;FOLD SLIN P513 Vel=1 m/s CPDAT513 Tool[4]:Microflown3D Base[0];%{PE}
;FOLD Parameters ;%{h}
;Params IlfProvider=kukaroboter.basistech.inlineforms.movement.spline; Kuka.IsGlobalPoint=False; Kuka.PointName=P513; Kuka.BlendingEnabled=False; Kuka.MoveDataName=CPDAT513; Kuka.VelocityPath=1.000; Kuka.VelocityFieldEnabled=True; Kuka.ColDetectFieldEnabled=True; Kuka.CurrentCDSetIndex=0; Kuka.MovementParameterFieldEnabled=True; IlfCommand=SLIN
;ENDFOLD
SLIN XP513 WITH $VEL = SVEL_CP(2.0, , LCPDAT513),$TOOL = STOOL2(FP513),$BASE = SBASE(FP513.BASE_NO),$IPO_MODE = SIPO_MODE(FP513.IPO_FRAME),$LOAD = SLOAD(FP513.TOOL_NO),$ACC = SACC_CP(LCPDAT513),$ORI_TYPE = SORI_TYP(LCPDAT513),$APO = SAPO(LCPDAT513),$JERK = SJERK(LCPDAT513),$COLLMON_TOL_PRO[1] = USE_CM_PRO_VALUES(0)
;ENDFOLD

;FOLD SLIN P514 Vel=1 m/s CPDAT514 Tool[4]:Microflown3D Base[0];%{PE}
;FOLD Parameters ;%{h}
;Params IlfProvider=kukaroboter.basistech.inlineforms.movement.spline; Kuka.IsGlobalPoint=False; Kuka.PointName=P514; Kuka.BlendingEnabled=False; Kuka.MoveDataName=CPDAT514; Kuka.VelocityPath=1.000; Kuka.VelocityFieldEnabled=True; Kuka.ColDetectFieldEnabled=True; Kuka.CurrentCDSetIndex=0; Kuka.MovementParameterFieldEnabled=True; IlfCommand=SLIN
;ENDFOLD
SLIN XP514 WITH $VEL = SVEL_CP(2.0, , LCPDAT514),$TOOL = STOOL2(FP514),$BASE = SBASE(FP514.BASE_NO),$IPO_MODE = SIPO_MODE(FP514.IPO_FRAME),$LOAD = SLOAD(FP514.TOOL_NO),$ACC = SACC_CP(LCPDAT514),$ORI_TYPE = SORI_TYP(LCPDAT514),$APO = SAPO(LCPDAT514),$JERK = SJERK(LCPDAT514),$COLLMON_TOL_PRO[1] = USE_CM_PRO_VALUES(0)
;ENDFOLD

;FOLD SLIN P515 Vel=1 m/s CPDAT515 Tool[4]:Microflown3D Base[0];%{PE}
;FOLD Parameters ;%{h}
;Params IlfProvider=kukaroboter.basistech.inlineforms.movement.spline; Kuka.IsGlobalPoint=False; Kuka.PointName=P515; Kuka.BlendingEnabled=False; Kuka.MoveDataName=CPDAT515; Kuka.VelocityPath=1.000; Kuka.VelocityFieldEnabled=True; Kuka.ColDetectFieldEnabled=True; Kuka.CurrentCDSetIndex=0; Kuka.MovementParameterFieldEnabled=True; IlfCommand=SLIN
;ENDFOLD
SLIN XP515 WITH $VEL = SVEL_CP(2.0, , LCPDAT515),$TOOL = STOOL2(FP515),$BASE = SBASE(FP515.BASE_NO),$IPO_MODE = SIPO_MODE(FP515.IPO_FRAME),$LOAD = SLOAD(FP515.TOOL_NO),$ACC = SACC_CP(LCPDAT515),$ORI_TYPE = SORI_TYP(LCPDAT515),$APO = SAPO(LCPDAT515),$JERK = SJERK(LCPDAT515),$COLLMON_TOL_PRO[1] = USE_CM_PRO_VALUES(0)
;ENDFOLD

;FOLD SLIN P516 Vel=1 m/s CPDAT516 Tool[4]:Microflown3D Base[0];%{PE}
;FOLD Parameters ;%{h}
;Params IlfProvider=kukaroboter.basistech.inlineforms.movement.spline; Kuka.IsGlobalPoint=False; Kuka.PointName=P516; Kuka.BlendingEnabled=False; Kuka.MoveDataName=CPDAT516; Kuka.VelocityPath=1.000; Kuka.VelocityFieldEnabled=True; Kuka.ColDetectFieldEnabled=True; Kuka.CurrentCDSetIndex=0; Kuka.MovementParameterFieldEnabled=True; IlfCommand=SLIN
;ENDFOLD
SLIN XP516 WITH $VEL = SVEL_CP(2.0, , LCPDAT516),$TOOL = STOOL2(FP516),$BASE = SBASE(FP516.BASE_NO),$IPO_MODE = SIPO_MODE(FP516.IPO_FRAME),$LOAD = SLOAD(FP516.TOOL_NO),$ACC = SACC_CP(LCPDAT516),$ORI_TYPE = SORI_TYP(LCPDAT516),$APO = SAPO(LCPDAT516),$JERK = SJERK(LCPDAT516),$COLLMON_TOL_PRO[1] = USE_CM_PRO_VALUES(0)
;ENDFOLD

;FOLD SLIN P517 Vel=1 m/s CPDAT517 Tool[4]:Microflown3D Base[0];%{PE}
;FOLD Parameters ;%{h}
;Params IlfProvider=kukaroboter.basistech.inlineforms.movement.spline; Kuka.IsGlobalPoint=False; Kuka.PointName=P517; Kuka.BlendingEnabled=False; Kuka.MoveDataName=CPDAT517; Kuka.VelocityPath=1.000; Kuka.VelocityFieldEnabled=True; Kuka.ColDetectFieldEnabled=True; Kuka.CurrentCDSetIndex=0; Kuka.MovementParameterFieldEnabled=True; IlfCommand=SLIN
;ENDFOLD
SLIN XP517 WITH $VEL = SVEL_CP(2.0, , LCPDAT517),$TOOL = STOOL2(FP517),$BASE = SBASE(FP517.BASE_NO),$IPO_MODE = SIPO_MODE(FP517.IPO_FRAME),$LOAD = SLOAD(FP517.TOOL_NO),$ACC = SACC_CP(LCPDAT517),$ORI_TYPE = SORI_TYP(LCPDAT517),$APO = SAPO(LCPDAT517),$JERK = SJERK(LCPDAT517),$COLLMON_TOL_PRO[1] = USE_CM_PRO_VALUES(0)
;ENDFOLD

;FOLD SLIN P518 Vel=1 m/s CPDAT518 Tool[4]:Microflown3D Base[0];%{PE}
;FOLD Parameters ;%{h}
;Params IlfProvider=kukaroboter.basistech.inlineforms.movement.spline; Kuka.IsGlobalPoint=False; Kuka.PointName=P518; Kuka.BlendingEnabled=False; Kuka.MoveDataName=CPDAT518; Kuka.VelocityPath=1.000; Kuka.VelocityFieldEnabled=True; Kuka.ColDetectFieldEnabled=True; Kuka.CurrentCDSetIndex=0; Kuka.MovementParameterFieldEnabled=True; IlfCommand=SLIN
;ENDFOLD
SLIN XP518 WITH $VEL = SVEL_CP(2.0, , LCPDAT518),$TOOL = STOOL2(FP518),$BASE = SBASE(FP518.BASE_NO),$IPO_MODE = SIPO_MODE(FP518.IPO_FRAME),$LOAD = SLOAD(FP518.TOOL_NO),$ACC = SACC_CP(LCPDAT518),$ORI_TYPE = SORI_TYP(LCPDAT518),$APO = SAPO(LCPDAT518),$JERK = SJERK(LCPDAT518),$COLLMON_TOL_PRO[1] = USE_CM_PRO_VALUES(0)
;ENDFOLD

;FOLD SLIN P519 Vel=1 m/s CPDAT519 Tool[4]:Microflown3D Base[0];%{PE}
;FOLD Parameters ;%{h}
;Params IlfProvider=kukaroboter.basistech.inlineforms.movement.spline; Kuka.IsGlobalPoint=False; Kuka.PointName=P519; Kuka.BlendingEnabled=False; Kuka.MoveDataName=CPDAT519; Kuka.VelocityPath=1.000; Kuka.VelocityFieldEnabled=True; Kuka.ColDetectFieldEnabled=True; Kuka.CurrentCDSetIndex=0; Kuka.MovementParameterFieldEnabled=True; IlfCommand=SLIN
;ENDFOLD
SLIN XP519 WITH $VEL = SVEL_CP(2.0, , LCPDAT519),$TOOL = STOOL2(FP519),$BASE = SBASE(FP519.BASE_NO),$IPO_MODE = SIPO_MODE(FP519.IPO_FRAME),$LOAD = SLOAD(FP519.TOOL_NO),$ACC = SACC_CP(LCPDAT519),$ORI_TYPE = SORI_TYP(LCPDAT519),$APO = SAPO(LCPDAT519),$JERK = SJERK(LCPDAT519),$COLLMON_TOL_PRO[1] = USE_CM_PRO_VALUES(0)
;ENDFOLD

;FOLD SLIN P520 Vel=1 m/s CPDAT520 Tool[4]:Microflown3D Base[0];%{PE}
;FOLD Parameters ;%{h}
;Params IlfProvider=kukaroboter.basistech.inlineforms.movement.spline; Kuka.IsGlobalPoint=False; Kuka.PointName=P520; Kuka.BlendingEnabled=False; Kuka.MoveDataName=CPDAT520; Kuka.VelocityPath=1.000; Kuka.VelocityFieldEnabled=True; Kuka.ColDetectFieldEnabled=True; Kuka.CurrentCDSetIndex=0; Kuka.MovementParameterFieldEnabled=True; IlfCommand=SLIN
;ENDFOLD
SLIN XP520 WITH $VEL = SVEL_CP(2.0, , LCPDAT520),$TOOL = STOOL2(FP520),$BASE = SBASE(FP520.BASE_NO),$IPO_MODE = SIPO_MODE(FP520.IPO_FRAME),$LOAD = SLOAD(FP520.TOOL_NO),$ACC = SACC_CP(LCPDAT520),$ORI_TYPE = SORI_TYP(LCPDAT520),$APO = SAPO(LCPDAT520),$JERK = SJERK(LCPDAT520),$COLLMON_TOL_PRO[1] = USE_CM_PRO_VALUES(0)
;ENDFOLD

;FOLD SLIN P521 Vel=1 m/s CPDAT521 Tool[4]:Microflown3D Base[0];%{PE}
;FOLD Parameters ;%{h}
;Params IlfProvider=kukaroboter.basistech.inlineforms.movement.spline; Kuka.IsGlobalPoint=False; Kuka.PointName=P521; Kuka.BlendingEnabled=False; Kuka.MoveDataName=CPDAT521; Kuka.VelocityPath=1.000; Kuka.VelocityFieldEnabled=True; Kuka.ColDetectFieldEnabled=True; Kuka.CurrentCDSetIndex=0; Kuka.MovementParameterFieldEnabled=True; IlfCommand=SLIN
;ENDFOLD
SLIN XP521 WITH $VEL = SVEL_CP(2.0, , LCPDAT521),$TOOL = STOOL2(FP521),$BASE = SBASE(FP521.BASE_NO),$IPO_MODE = SIPO_MODE(FP521.IPO_FRAME),$LOAD = SLOAD(FP521.TOOL_NO),$ACC = SACC_CP(LCPDAT521),$ORI_TYPE = SORI_TYP(LCPDAT521),$APO = SAPO(LCPDAT521),$JERK = SJERK(LCPDAT521),$COLLMON_TOL_PRO[1] = USE_CM_PRO_VALUES(0)
;ENDFOLD

;FOLD SLIN P522 Vel=1 m/s CPDAT522 Tool[4]:Microflown3D Base[0];%{PE}
;FOLD Parameters ;%{h}
;Params IlfProvider=kukaroboter.basistech.inlineforms.movement.spline; Kuka.IsGlobalPoint=False; Kuka.PointName=P522; Kuka.BlendingEnabled=False; Kuka.MoveDataName=CPDAT522; Kuka.VelocityPath=1.000; Kuka.VelocityFieldEnabled=True; Kuka.ColDetectFieldEnabled=True; Kuka.CurrentCDSetIndex=0; Kuka.MovementParameterFieldEnabled=True; IlfCommand=SLIN
;ENDFOLD
SLIN XP522 WITH $VEL = SVEL_CP(2.0, , LCPDAT522),$TOOL = STOOL2(FP522),$BASE = SBASE(FP522.BASE_NO),$IPO_MODE = SIPO_MODE(FP522.IPO_FRAME),$LOAD = SLOAD(FP522.TOOL_NO),$ACC = SACC_CP(LCPDAT522),$ORI_TYPE = SORI_TYP(LCPDAT522),$APO = SAPO(LCPDAT522),$JERK = SJERK(LCPDAT522),$COLLMON_TOL_PRO[1] = USE_CM_PRO_VALUES(0)
;ENDFOLD

;FOLD SLIN P523 Vel=1 m/s CPDAT523 Tool[4]:Microflown3D Base[0];%{PE}
;FOLD Parameters ;%{h}
;Params IlfProvider=kukaroboter.basistech.inlineforms.movement.spline; Kuka.IsGlobalPoint=False; Kuka.PointName=P523; Kuka.BlendingEnabled=False; Kuka.MoveDataName=CPDAT523; Kuka.VelocityPath=1.000; Kuka.VelocityFieldEnabled=True; Kuka.ColDetectFieldEnabled=True; Kuka.CurrentCDSetIndex=0; Kuka.MovementParameterFieldEnabled=True; IlfCommand=SLIN
;ENDFOLD
SLIN XP523 WITH $VEL = SVEL_CP(2.0, , LCPDAT523),$TOOL = STOOL2(FP523),$BASE = SBASE(FP523.BASE_NO),$IPO_MODE = SIPO_MODE(FP523.IPO_FRAME),$LOAD = SLOAD(FP523.TOOL_NO),$ACC = SACC_CP(LCPDAT523),$ORI_TYPE = SORI_TYP(LCPDAT523),$APO = SAPO(LCPDAT523),$JERK = SJERK(LCPDAT523),$COLLMON_TOL_PRO[1] = USE_CM_PRO_VALUES(0)
;ENDFOLD

;FOLD SLIN P524 Vel=1 m/s CPDAT524 Tool[4]:Microflown3D Base[0];%{PE}
;FOLD Parameters ;%{h}
;Params IlfProvider=kukaroboter.basistech.inlineforms.movement.spline; Kuka.IsGlobalPoint=False; Kuka.PointName=P524; Kuka.BlendingEnabled=False; Kuka.MoveDataName=CPDAT524; Kuka.VelocityPath=1.000; Kuka.VelocityFieldEnabled=True; Kuka.ColDetectFieldEnabled=True; Kuka.CurrentCDSetIndex=0; Kuka.MovementParameterFieldEnabled=True; IlfCommand=SLIN
;ENDFOLD
SLIN XP524 WITH $VEL = SVEL_CP(2.0, , LCPDAT524),$TOOL = STOOL2(FP524),$BASE = SBASE(FP524.BASE_NO),$IPO_MODE = SIPO_MODE(FP524.IPO_FRAME),$LOAD = SLOAD(FP524.TOOL_NO),$ACC = SACC_CP(LCPDAT524),$ORI_TYPE = SORI_TYP(LCPDAT524),$APO = SAPO(LCPDAT524),$JERK = SJERK(LCPDAT524),$COLLMON_TOL_PRO[1] = USE_CM_PRO_VALUES(0)
;ENDFOLD

;FOLD SLIN P525 Vel=1 m/s CPDAT525 Tool[4]:Microflown3D Base[0];%{PE}
;FOLD Parameters ;%{h}
;Params IlfProvider=kukaroboter.basistech.inlineforms.movement.spline; Kuka.IsGlobalPoint=False; Kuka.PointName=P525; Kuka.BlendingEnabled=False; Kuka.MoveDataName=CPDAT525; Kuka.VelocityPath=1.000; Kuka.VelocityFieldEnabled=True; Kuka.ColDetectFieldEnabled=True; Kuka.CurrentCDSetIndex=0; Kuka.MovementParameterFieldEnabled=True; IlfCommand=SLIN
;ENDFOLD
SLIN XP525 WITH $VEL = SVEL_CP(2.0, , LCPDAT525),$TOOL = STOOL2(FP525),$BASE = SBASE(FP525.BASE_NO),$IPO_MODE = SIPO_MODE(FP525.IPO_FRAME),$LOAD = SLOAD(FP525.TOOL_NO),$ACC = SACC_CP(LCPDAT525),$ORI_TYPE = SORI_TYP(LCPDAT525),$APO = SAPO(LCPDAT525),$JERK = SJERK(LCPDAT525),$COLLMON_TOL_PRO[1] = USE_CM_PRO_VALUES(0)
;ENDFOLD

;FOLD SLIN P526 Vel=1 m/s CPDAT526 Tool[4]:Microflown3D Base[0];%{PE}
;FOLD Parameters ;%{h}
;Params IlfProvider=kukaroboter.basistech.inlineforms.movement.spline; Kuka.IsGlobalPoint=False; Kuka.PointName=P526; Kuka.BlendingEnabled=False; Kuka.MoveDataName=CPDAT526; Kuka.VelocityPath=1.000; Kuka.VelocityFieldEnabled=True; Kuka.ColDetectFieldEnabled=True; Kuka.CurrentCDSetIndex=0; Kuka.MovementParameterFieldEnabled=True; IlfCommand=SLIN
;ENDFOLD
SLIN XP526 WITH $VEL = SVEL_CP(2.0, , LCPDAT526),$TOOL = STOOL2(FP526),$BASE = SBASE(FP526.BASE_NO),$IPO_MODE = SIPO_MODE(FP526.IPO_FRAME),$LOAD = SLOAD(FP526.TOOL_NO),$ACC = SACC_CP(LCPDAT526),$ORI_TYPE = SORI_TYP(LCPDAT526),$APO = SAPO(LCPDAT526),$JERK = SJERK(LCPDAT526),$COLLMON_TOL_PRO[1] = USE_CM_PRO_VALUES(0)
;ENDFOLD

;FOLD SLIN P527 Vel=1 m/s CPDAT527 Tool[4]:Microflown3D Base[0];%{PE}
;FOLD Parameters ;%{h}
;Params IlfProvider=kukaroboter.basistech.inlineforms.movement.spline; Kuka.IsGlobalPoint=False; Kuka.PointName=P527; Kuka.BlendingEnabled=False; Kuka.MoveDataName=CPDAT527; Kuka.VelocityPath=1.000; Kuka.VelocityFieldEnabled=True; Kuka.ColDetectFieldEnabled=True; Kuka.CurrentCDSetIndex=0; Kuka.MovementParameterFieldEnabled=True; IlfCommand=SLIN
;ENDFOLD
SLIN XP527 WITH $VEL = SVEL_CP(2.0, , LCPDAT527),$TOOL = STOOL2(FP527),$BASE = SBASE(FP527.BASE_NO),$IPO_MODE = SIPO_MODE(FP527.IPO_FRAME),$LOAD = SLOAD(FP527.TOOL_NO),$ACC = SACC_CP(LCPDAT527),$ORI_TYPE = SORI_TYP(LCPDAT527),$APO = SAPO(LCPDAT527),$JERK = SJERK(LCPDAT527),$COLLMON_TOL_PRO[1] = USE_CM_PRO_VALUES(0)
;ENDFOLD

;FOLD SLIN P528 Vel=1 m/s CPDAT528 Tool[4]:Microflown3D Base[0];%{PE}
;FOLD Parameters ;%{h}
;Params IlfProvider=kukaroboter.basistech.inlineforms.movement.spline; Kuka.IsGlobalPoint=False; Kuka.PointName=P528; Kuka.BlendingEnabled=False; Kuka.MoveDataName=CPDAT528; Kuka.VelocityPath=1.000; Kuka.VelocityFieldEnabled=True; Kuka.ColDetectFieldEnabled=True; Kuka.CurrentCDSetIndex=0; Kuka.MovementParameterFieldEnabled=True; IlfCommand=SLIN
;ENDFOLD
SLIN XP528 WITH $VEL = SVEL_CP(2.0, , LCPDAT528),$TOOL = STOOL2(FP528),$BASE = SBASE(FP528.BASE_NO),$IPO_MODE = SIPO_MODE(FP528.IPO_FRAME),$LOAD = SLOAD(FP528.TOOL_NO),$ACC = SACC_CP(LCPDAT528),$ORI_TYPE = SORI_TYP(LCPDAT528),$APO = SAPO(LCPDAT528),$JERK = SJERK(LCPDAT528),$COLLMON_TOL_PRO[1] = USE_CM_PRO_VALUES(0)
;ENDFOLD

;FOLD SLIN P529 Vel=1 m/s CPDAT529 Tool[4]:Microflown3D Base[0];%{PE}
;FOLD Parameters ;%{h}
;Params IlfProvider=kukaroboter.basistech.inlineforms.movement.spline; Kuka.IsGlobalPoint=False; Kuka.PointName=P529; Kuka.BlendingEnabled=False; Kuka.MoveDataName=CPDAT529; Kuka.VelocityPath=1.000; Kuka.VelocityFieldEnabled=True; Kuka.ColDetectFieldEnabled=True; Kuka.CurrentCDSetIndex=0; Kuka.MovementParameterFieldEnabled=True; IlfCommand=SLIN
;ENDFOLD
SLIN XP529 WITH $VEL = SVEL_CP(2.0, , LCPDAT529),$TOOL = STOOL2(FP529),$BASE = SBASE(FP529.BASE_NO),$IPO_MODE = SIPO_MODE(FP529.IPO_FRAME),$LOAD = SLOAD(FP529.TOOL_NO),$ACC = SACC_CP(LCPDAT529),$ORI_TYPE = SORI_TYP(LCPDAT529),$APO = SAPO(LCPDAT529),$JERK = SJERK(LCPDAT529),$COLLMON_TOL_PRO[1] = USE_CM_PRO_VALUES(0)
;ENDFOLD

;FOLD SLIN P530 Vel=1 m/s CPDAT530 Tool[4]:Microflown3D Base[0];%{PE}
;FOLD Parameters ;%{h}
;Params IlfProvider=kukaroboter.basistech.inlineforms.movement.spline; Kuka.IsGlobalPoint=False; Kuka.PointName=P530; Kuka.BlendingEnabled=False; Kuka.MoveDataName=CPDAT530; Kuka.VelocityPath=1.000; Kuka.VelocityFieldEnabled=True; Kuka.ColDetectFieldEnabled=True; Kuka.CurrentCDSetIndex=0; Kuka.MovementParameterFieldEnabled=True; IlfCommand=SLIN
;ENDFOLD
SLIN XP530 WITH $VEL = SVEL_CP(2.0, , LCPDAT530),$TOOL = STOOL2(FP530),$BASE = SBASE(FP530.BASE_NO),$IPO_MODE = SIPO_MODE(FP530.IPO_FRAME),$LOAD = SLOAD(FP530.TOOL_NO),$ACC = SACC_CP(LCPDAT530),$ORI_TYPE = SORI_TYP(LCPDAT530),$APO = SAPO(LCPDAT530),$JERK = SJERK(LCPDAT530),$COLLMON_TOL_PRO[1] = USE_CM_PRO_VALUES(0)
;ENDFOLD

;FOLD SLIN P531 Vel=1 m/s CPDAT531 Tool[4]:Microflown3D Base[0];%{PE}
;FOLD Parameters ;%{h}
;Params IlfProvider=kukaroboter.basistech.inlineforms.movement.spline; Kuka.IsGlobalPoint=False; Kuka.PointName=P531; Kuka.BlendingEnabled=False; Kuka.MoveDataName=CPDAT531; Kuka.VelocityPath=1.000; Kuka.VelocityFieldEnabled=True; Kuka.ColDetectFieldEnabled=True; Kuka.CurrentCDSetIndex=0; Kuka.MovementParameterFieldEnabled=True; IlfCommand=SLIN
;ENDFOLD
SLIN XP531 WITH $VEL = SVEL_CP(2.0, , LCPDAT531),$TOOL = STOOL2(FP531),$BASE = SBASE(FP531.BASE_NO),$IPO_MODE = SIPO_MODE(FP531.IPO_FRAME),$LOAD = SLOAD(FP531.TOOL_NO),$ACC = SACC_CP(LCPDAT531),$ORI_TYPE = SORI_TYP(LCPDAT531),$APO = SAPO(LCPDAT531),$JERK = SJERK(LCPDAT531),$COLLMON_TOL_PRO[1] = USE_CM_PRO_VALUES(0)
;ENDFOLD

;FOLD SLIN P532 Vel=1 m/s CPDAT532 Tool[4]:Microflown3D Base[0];%{PE}
;FOLD Parameters ;%{h}
;Params IlfProvider=kukaroboter.basistech.inlineforms.movement.spline; Kuka.IsGlobalPoint=False; Kuka.PointName=P532; Kuka.BlendingEnabled=False; Kuka.MoveDataName=CPDAT532; Kuka.VelocityPath=1.000; Kuka.VelocityFieldEnabled=True; Kuka.ColDetectFieldEnabled=True; Kuka.CurrentCDSetIndex=0; Kuka.MovementParameterFieldEnabled=True; IlfCommand=SLIN
;ENDFOLD
SLIN XP532 WITH $VEL = SVEL_CP(2.0, , LCPDAT532),$TOOL = STOOL2(FP532),$BASE = SBASE(FP532.BASE_NO),$IPO_MODE = SIPO_MODE(FP532.IPO_FRAME),$LOAD = SLOAD(FP532.TOOL_NO),$ACC = SACC_CP(LCPDAT532),$ORI_TYPE = SORI_TYP(LCPDAT532),$APO = SAPO(LCPDAT532),$JERK = SJERK(LCPDAT532),$COLLMON_TOL_PRO[1] = USE_CM_PRO_VALUES(0)
;ENDFOLD

;FOLD SLIN P533 Vel=1 m/s CPDAT533 Tool[4]:Microflown3D Base[0];%{PE}
;FOLD Parameters ;%{h}
;Params IlfProvider=kukaroboter.basistech.inlineforms.movement.spline; Kuka.IsGlobalPoint=False; Kuka.PointName=P533; Kuka.BlendingEnabled=False; Kuka.MoveDataName=CPDAT533; Kuka.VelocityPath=1.000; Kuka.VelocityFieldEnabled=True; Kuka.ColDetectFieldEnabled=True; Kuka.CurrentCDSetIndex=0; Kuka.MovementParameterFieldEnabled=True; IlfCommand=SLIN
;ENDFOLD
SLIN XP533 WITH $VEL = SVEL_CP(2.0, , LCPDAT533),$TOOL = STOOL2(FP533),$BASE = SBASE(FP533.BASE_NO),$IPO_MODE = SIPO_MODE(FP533.IPO_FRAME),$LOAD = SLOAD(FP533.TOOL_NO),$ACC = SACC_CP(LCPDAT533),$ORI_TYPE = SORI_TYP(LCPDAT533),$APO = SAPO(LCPDAT533),$JERK = SJERK(LCPDAT533),$COLLMON_TOL_PRO[1] = USE_CM_PRO_VALUES(0)
;ENDFOLD

;FOLD SLIN P534 Vel=1 m/s CPDAT534 Tool[4]:Microflown3D Base[0];%{PE}
;FOLD Parameters ;%{h}
;Params IlfProvider=kukaroboter.basistech.inlineforms.movement.spline; Kuka.IsGlobalPoint=False; Kuka.PointName=P534; Kuka.BlendingEnabled=False; Kuka.MoveDataName=CPDAT534; Kuka.VelocityPath=1.000; Kuka.VelocityFieldEnabled=True; Kuka.ColDetectFieldEnabled=True; Kuka.CurrentCDSetIndex=0; Kuka.MovementParameterFieldEnabled=True; IlfCommand=SLIN
;ENDFOLD
SLIN XP534 WITH $VEL = SVEL_CP(2.0, , LCPDAT534),$TOOL = STOOL2(FP534),$BASE = SBASE(FP534.BASE_NO),$IPO_MODE = SIPO_MODE(FP534.IPO_FRAME),$LOAD = SLOAD(FP534.TOOL_NO),$ACC = SACC_CP(LCPDAT534),$ORI_TYPE = SORI_TYP(LCPDAT534),$APO = SAPO(LCPDAT534),$JERK = SJERK(LCPDAT534),$COLLMON_TOL_PRO[1] = USE_CM_PRO_VALUES(0)
;ENDFOLD

;FOLD SLIN P535 Vel=1 m/s CPDAT535 Tool[4]:Microflown3D Base[0];%{PE}
;FOLD Parameters ;%{h}
;Params IlfProvider=kukaroboter.basistech.inlineforms.movement.spline; Kuka.IsGlobalPoint=False; Kuka.PointName=P535; Kuka.BlendingEnabled=False; Kuka.MoveDataName=CPDAT535; Kuka.VelocityPath=1.000; Kuka.VelocityFieldEnabled=True; Kuka.ColDetectFieldEnabled=True; Kuka.CurrentCDSetIndex=0; Kuka.MovementParameterFieldEnabled=True; IlfCommand=SLIN
;ENDFOLD
SLIN XP535 WITH $VEL = SVEL_CP(2.0, , LCPDAT535),$TOOL = STOOL2(FP535),$BASE = SBASE(FP535.BASE_NO),$IPO_MODE = SIPO_MODE(FP535.IPO_FRAME),$LOAD = SLOAD(FP535.TOOL_NO),$ACC = SACC_CP(LCPDAT535),$ORI_TYPE = SORI_TYP(LCPDAT535),$APO = SAPO(LCPDAT535),$JERK = SJERK(LCPDAT535),$COLLMON_TOL_PRO[1] = USE_CM_PRO_VALUES(0)
;ENDFOLD

;FOLD SLIN P536 Vel=1 m/s CPDAT536 Tool[4]:Microflown3D Base[0];%{PE}
;FOLD Parameters ;%{h}
;Params IlfProvider=kukaroboter.basistech.inlineforms.movement.spline; Kuka.IsGlobalPoint=False; Kuka.PointName=P536; Kuka.BlendingEnabled=False; Kuka.MoveDataName=CPDAT536; Kuka.VelocityPath=1.000; Kuka.VelocityFieldEnabled=True; Kuka.ColDetectFieldEnabled=True; Kuka.CurrentCDSetIndex=0; Kuka.MovementParameterFieldEnabled=True; IlfCommand=SLIN
;ENDFOLD
SLIN XP536 WITH $VEL = SVEL_CP(2.0, , LCPDAT536),$TOOL = STOOL2(FP536),$BASE = SBASE(FP536.BASE_NO),$IPO_MODE = SIPO_MODE(FP536.IPO_FRAME),$LOAD = SLOAD(FP536.TOOL_NO),$ACC = SACC_CP(LCPDAT536),$ORI_TYPE = SORI_TYP(LCPDAT536),$APO = SAPO(LCPDAT536),$JERK = SJERK(LCPDAT536),$COLLMON_TOL_PRO[1] = USE_CM_PRO_VALUES(0)
;ENDFOLD

;FOLD SLIN P537 Vel=1 m/s CPDAT537 Tool[4]:Microflown3D Base[0];%{PE}
;FOLD Parameters ;%{h}
;Params IlfProvider=kukaroboter.basistech.inlineforms.movement.spline; Kuka.IsGlobalPoint=False; Kuka.PointName=P537; Kuka.BlendingEnabled=False; Kuka.MoveDataName=CPDAT537; Kuka.VelocityPath=1.000; Kuka.VelocityFieldEnabled=True; Kuka.ColDetectFieldEnabled=True; Kuka.CurrentCDSetIndex=0; Kuka.MovementParameterFieldEnabled=True; IlfCommand=SLIN
;ENDFOLD
SLIN XP537 WITH $VEL = SVEL_CP(2.0, , LCPDAT537),$TOOL = STOOL2(FP537),$BASE = SBASE(FP537.BASE_NO),$IPO_MODE = SIPO_MODE(FP537.IPO_FRAME),$LOAD = SLOAD(FP537.TOOL_NO),$ACC = SACC_CP(LCPDAT537),$ORI_TYPE = SORI_TYP(LCPDAT537),$APO = SAPO(LCPDAT537),$JERK = SJERK(LCPDAT537),$COLLMON_TOL_PRO[1] = USE_CM_PRO_VALUES(0)
;ENDFOLD

;FOLD SLIN P538 Vel=1 m/s CPDAT538 Tool[4]:Microflown3D Base[0];%{PE}
;FOLD Parameters ;%{h}
;Params IlfProvider=kukaroboter.basistech.inlineforms.movement.spline; Kuka.IsGlobalPoint=False; Kuka.PointName=P538; Kuka.BlendingEnabled=False; Kuka.MoveDataName=CPDAT538; Kuka.VelocityPath=1.000; Kuka.VelocityFieldEnabled=True; Kuka.ColDetectFieldEnabled=True; Kuka.CurrentCDSetIndex=0; Kuka.MovementParameterFieldEnabled=True; IlfCommand=SLIN
;ENDFOLD
SLIN XP538 WITH $VEL = SVEL_CP(2.0, , LCPDAT538),$TOOL = STOOL2(FP538),$BASE = SBASE(FP538.BASE_NO),$IPO_MODE = SIPO_MODE(FP538.IPO_FRAME),$LOAD = SLOAD(FP538.TOOL_NO),$ACC = SACC_CP(LCPDAT538),$ORI_TYPE = SORI_TYP(LCPDAT538),$APO = SAPO(LCPDAT538),$JERK = SJERK(LCPDAT538),$COLLMON_TOL_PRO[1] = USE_CM_PRO_VALUES(0)
;ENDFOLD

;FOLD SLIN P539 Vel=1 m/s CPDAT539 Tool[4]:Microflown3D Base[0];%{PE}
;FOLD Parameters ;%{h}
;Params IlfProvider=kukaroboter.basistech.inlineforms.movement.spline; Kuka.IsGlobalPoint=False; Kuka.PointName=P539; Kuka.BlendingEnabled=False; Kuka.MoveDataName=CPDAT539; Kuka.VelocityPath=1.000; Kuka.VelocityFieldEnabled=True; Kuka.ColDetectFieldEnabled=True; Kuka.CurrentCDSetIndex=0; Kuka.MovementParameterFieldEnabled=True; IlfCommand=SLIN
;ENDFOLD
SLIN XP539 WITH $VEL = SVEL_CP(2.0, , LCPDAT539),$TOOL = STOOL2(FP539),$BASE = SBASE(FP539.BASE_NO),$IPO_MODE = SIPO_MODE(FP539.IPO_FRAME),$LOAD = SLOAD(FP539.TOOL_NO),$ACC = SACC_CP(LCPDAT539),$ORI_TYPE = SORI_TYP(LCPDAT539),$APO = SAPO(LCPDAT539),$JERK = SJERK(LCPDAT539),$COLLMON_TOL_PRO[1] = USE_CM_PRO_VALUES(0)
;ENDFOLD

;FOLD SLIN P540 Vel=1 m/s CPDAT540 Tool[4]:Microflown3D Base[0];%{PE}
;FOLD Parameters ;%{h}
;Params IlfProvider=kukaroboter.basistech.inlineforms.movement.spline; Kuka.IsGlobalPoint=False; Kuka.PointName=P540; Kuka.BlendingEnabled=False; Kuka.MoveDataName=CPDAT540; Kuka.VelocityPath=1.000; Kuka.VelocityFieldEnabled=True; Kuka.ColDetectFieldEnabled=True; Kuka.CurrentCDSetIndex=0; Kuka.MovementParameterFieldEnabled=True; IlfCommand=SLIN
;ENDFOLD
SLIN XP540 WITH $VEL = SVEL_CP(2.0, , LCPDAT540),$TOOL = STOOL2(FP540),$BASE = SBASE(FP540.BASE_NO),$IPO_MODE = SIPO_MODE(FP540.IPO_FRAME),$LOAD = SLOAD(FP540.TOOL_NO),$ACC = SACC_CP(LCPDAT540),$ORI_TYPE = SORI_TYP(LCPDAT540),$APO = SAPO(LCPDAT540),$JERK = SJERK(LCPDAT540),$COLLMON_TOL_PRO[1] = USE_CM_PRO_VALUES(0)
;ENDFOLD

;FOLD SLIN P541 Vel=1 m/s CPDAT541 Tool[4]:Microflown3D Base[0];%{PE}
;FOLD Parameters ;%{h}
;Params IlfProvider=kukaroboter.basistech.inlineforms.movement.spline; Kuka.IsGlobalPoint=False; Kuka.PointName=P541; Kuka.BlendingEnabled=False; Kuka.MoveDataName=CPDAT541; Kuka.VelocityPath=1.000; Kuka.VelocityFieldEnabled=True; Kuka.ColDetectFieldEnabled=True; Kuka.CurrentCDSetIndex=0; Kuka.MovementParameterFieldEnabled=True; IlfCommand=SLIN
;ENDFOLD
SLIN XP541 WITH $VEL = SVEL_CP(2.0, , LCPDAT541),$TOOL = STOOL2(FP541),$BASE = SBASE(FP541.BASE_NO),$IPO_MODE = SIPO_MODE(FP541.IPO_FRAME),$LOAD = SLOAD(FP541.TOOL_NO),$ACC = SACC_CP(LCPDAT541),$ORI_TYPE = SORI_TYP(LCPDAT541),$APO = SAPO(LCPDAT541),$JERK = SJERK(LCPDAT541),$COLLMON_TOL_PRO[1] = USE_CM_PRO_VALUES(0)
;ENDFOLD

;FOLD SLIN P542 Vel=1 m/s CPDAT542 Tool[4]:Microflown3D Base[0];%{PE}
;FOLD Parameters ;%{h}
;Params IlfProvider=kukaroboter.basistech.inlineforms.movement.spline; Kuka.IsGlobalPoint=False; Kuka.PointName=P542; Kuka.BlendingEnabled=False; Kuka.MoveDataName=CPDAT542; Kuka.VelocityPath=1.000; Kuka.VelocityFieldEnabled=True; Kuka.ColDetectFieldEnabled=True; Kuka.CurrentCDSetIndex=0; Kuka.MovementParameterFieldEnabled=True; IlfCommand=SLIN
;ENDFOLD
SLIN XP542 WITH $VEL = SVEL_CP(2.0, , LCPDAT542),$TOOL = STOOL2(FP542),$BASE = SBASE(FP542.BASE_NO),$IPO_MODE = SIPO_MODE(FP542.IPO_FRAME),$LOAD = SLOAD(FP542.TOOL_NO),$ACC = SACC_CP(LCPDAT542),$ORI_TYPE = SORI_TYP(LCPDAT542),$APO = SAPO(LCPDAT542),$JERK = SJERK(LCPDAT542),$COLLMON_TOL_PRO[1] = USE_CM_PRO_VALUES(0)
;ENDFOLD

;FOLD SLIN P543 Vel=1 m/s CPDAT543 Tool[4]:Microflown3D Base[0];%{PE}
;FOLD Parameters ;%{h}
;Params IlfProvider=kukaroboter.basistech.inlineforms.movement.spline; Kuka.IsGlobalPoint=False; Kuka.PointName=P543; Kuka.BlendingEnabled=False; Kuka.MoveDataName=CPDAT543; Kuka.VelocityPath=1.000; Kuka.VelocityFieldEnabled=True; Kuka.ColDetectFieldEnabled=True; Kuka.CurrentCDSetIndex=0; Kuka.MovementParameterFieldEnabled=True; IlfCommand=SLIN
;ENDFOLD
SLIN XP543 WITH $VEL = SVEL_CP(2.0, , LCPDAT543),$TOOL = STOOL2(FP543),$BASE = SBASE(FP543.BASE_NO),$IPO_MODE = SIPO_MODE(FP543.IPO_FRAME),$LOAD = SLOAD(FP543.TOOL_NO),$ACC = SACC_CP(LCPDAT543),$ORI_TYPE = SORI_TYP(LCPDAT543),$APO = SAPO(LCPDAT543),$JERK = SJERK(LCPDAT543),$COLLMON_TOL_PRO[1] = USE_CM_PRO_VALUES(0)
;ENDFOLD

;FOLD SLIN P544 Vel=1 m/s CPDAT544 Tool[4]:Microflown3D Base[0];%{PE}
;FOLD Parameters ;%{h}
;Params IlfProvider=kukaroboter.basistech.inlineforms.movement.spline; Kuka.IsGlobalPoint=False; Kuka.PointName=P544; Kuka.BlendingEnabled=False; Kuka.MoveDataName=CPDAT544; Kuka.VelocityPath=1.000; Kuka.VelocityFieldEnabled=True; Kuka.ColDetectFieldEnabled=True; Kuka.CurrentCDSetIndex=0; Kuka.MovementParameterFieldEnabled=True; IlfCommand=SLIN
;ENDFOLD
SLIN XP544 WITH $VEL = SVEL_CP(2.0, , LCPDAT544),$TOOL = STOOL2(FP544),$BASE = SBASE(FP544.BASE_NO),$IPO_MODE = SIPO_MODE(FP544.IPO_FRAME),$LOAD = SLOAD(FP544.TOOL_NO),$ACC = SACC_CP(LCPDAT544),$ORI_TYPE = SORI_TYP(LCPDAT544),$APO = SAPO(LCPDAT544),$JERK = SJERK(LCPDAT544),$COLLMON_TOL_PRO[1] = USE_CM_PRO_VALUES(0)
;ENDFOLD

;FOLD SLIN P545 Vel=1 m/s CPDAT545 Tool[4]:Microflown3D Base[0];%{PE}
;FOLD Parameters ;%{h}
;Params IlfProvider=kukaroboter.basistech.inlineforms.movement.spline; Kuka.IsGlobalPoint=False; Kuka.PointName=P545; Kuka.BlendingEnabled=False; Kuka.MoveDataName=CPDAT545; Kuka.VelocityPath=1.000; Kuka.VelocityFieldEnabled=True; Kuka.ColDetectFieldEnabled=True; Kuka.CurrentCDSetIndex=0; Kuka.MovementParameterFieldEnabled=True; IlfCommand=SLIN
;ENDFOLD
SLIN XP545 WITH $VEL = SVEL_CP(2.0, , LCPDAT545),$TOOL = STOOL2(FP545),$BASE = SBASE(FP545.BASE_NO),$IPO_MODE = SIPO_MODE(FP545.IPO_FRAME),$LOAD = SLOAD(FP545.TOOL_NO),$ACC = SACC_CP(LCPDAT545),$ORI_TYPE = SORI_TYP(LCPDAT545),$APO = SAPO(LCPDAT545),$JERK = SJERK(LCPDAT545),$COLLMON_TOL_PRO[1] = USE_CM_PRO_VALUES(0)
;ENDFOLD

;FOLD SLIN P546 Vel=1 m/s CPDAT546 Tool[4]:Microflown3D Base[0];%{PE}
;FOLD Parameters ;%{h}
;Params IlfProvider=kukaroboter.basistech.inlineforms.movement.spline; Kuka.IsGlobalPoint=False; Kuka.PointName=P546; Kuka.BlendingEnabled=False; Kuka.MoveDataName=CPDAT546; Kuka.VelocityPath=1.000; Kuka.VelocityFieldEnabled=True; Kuka.ColDetectFieldEnabled=True; Kuka.CurrentCDSetIndex=0; Kuka.MovementParameterFieldEnabled=True; IlfCommand=SLIN
;ENDFOLD
SLIN XP546 WITH $VEL = SVEL_CP(2.0, , LCPDAT546),$TOOL = STOOL2(FP546),$BASE = SBASE(FP546.BASE_NO),$IPO_MODE = SIPO_MODE(FP546.IPO_FRAME),$LOAD = SLOAD(FP546.TOOL_NO),$ACC = SACC_CP(LCPDAT546),$ORI_TYPE = SORI_TYP(LCPDAT546),$APO = SAPO(LCPDAT546),$JERK = SJERK(LCPDAT546),$COLLMON_TOL_PRO[1] = USE_CM_PRO_VALUES(0)
;ENDFOLD

;FOLD SLIN P547 Vel=1 m/s CPDAT547 Tool[4]:Microflown3D Base[0];%{PE}
;FOLD Parameters ;%{h}
;Params IlfProvider=kukaroboter.basistech.inlineforms.movement.spline; Kuka.IsGlobalPoint=False; Kuka.PointName=P547; Kuka.BlendingEnabled=False; Kuka.MoveDataName=CPDAT547; Kuka.VelocityPath=1.000; Kuka.VelocityFieldEnabled=True; Kuka.ColDetectFieldEnabled=True; Kuka.CurrentCDSetIndex=0; Kuka.MovementParameterFieldEnabled=True; IlfCommand=SLIN
;ENDFOLD
SLIN XP547 WITH $VEL = SVEL_CP(2.0, , LCPDAT547),$TOOL = STOOL2(FP547),$BASE = SBASE(FP547.BASE_NO),$IPO_MODE = SIPO_MODE(FP547.IPO_FRAME),$LOAD = SLOAD(FP547.TOOL_NO),$ACC = SACC_CP(LCPDAT547),$ORI_TYPE = SORI_TYP(LCPDAT547),$APO = SAPO(LCPDAT547),$JERK = SJERK(LCPDAT547),$COLLMON_TOL_PRO[1] = USE_CM_PRO_VALUES(0)
;ENDFOLD

;FOLD SLIN P548 Vel=1 m/s CPDAT548 Tool[4]:Microflown3D Base[0];%{PE}
;FOLD Parameters ;%{h}
;Params IlfProvider=kukaroboter.basistech.inlineforms.movement.spline; Kuka.IsGlobalPoint=False; Kuka.PointName=P548; Kuka.BlendingEnabled=False; Kuka.MoveDataName=CPDAT548; Kuka.VelocityPath=1.000; Kuka.VelocityFieldEnabled=True; Kuka.ColDetectFieldEnabled=True; Kuka.CurrentCDSetIndex=0; Kuka.MovementParameterFieldEnabled=True; IlfCommand=SLIN
;ENDFOLD
SLIN XP548 WITH $VEL = SVEL_CP(2.0, , LCPDAT548),$TOOL = STOOL2(FP548),$BASE = SBASE(FP548.BASE_NO),$IPO_MODE = SIPO_MODE(FP548.IPO_FRAME),$LOAD = SLOAD(FP548.TOOL_NO),$ACC = SACC_CP(LCPDAT548),$ORI_TYPE = SORI_TYP(LCPDAT548),$APO = SAPO(LCPDAT548),$JERK = SJERK(LCPDAT548),$COLLMON_TOL_PRO[1] = USE_CM_PRO_VALUES(0)
;ENDFOLD

;FOLD SLIN P549 Vel=1 m/s CPDAT549 Tool[4]:Microflown3D Base[0];%{PE}
;FOLD Parameters ;%{h}
;Params IlfProvider=kukaroboter.basistech.inlineforms.movement.spline; Kuka.IsGlobalPoint=False; Kuka.PointName=P549; Kuka.BlendingEnabled=False; Kuka.MoveDataName=CPDAT549; Kuka.VelocityPath=1.000; Kuka.VelocityFieldEnabled=True; Kuka.ColDetectFieldEnabled=True; Kuka.CurrentCDSetIndex=0; Kuka.MovementParameterFieldEnabled=True; IlfCommand=SLIN
;ENDFOLD
SLIN XP549 WITH $VEL = SVEL_CP(2.0, , LCPDAT549),$TOOL = STOOL2(FP549),$BASE = SBASE(FP549.BASE_NO),$IPO_MODE = SIPO_MODE(FP549.IPO_FRAME),$LOAD = SLOAD(FP549.TOOL_NO),$ACC = SACC_CP(LCPDAT549),$ORI_TYPE = SORI_TYP(LCPDAT549),$APO = SAPO(LCPDAT549),$JERK = SJERK(LCPDAT549),$COLLMON_TOL_PRO[1] = USE_CM_PRO_VALUES(0)
;ENDFOLD

;FOLD SLIN P550 Vel=1 m/s CPDAT550 Tool[4]:Microflown3D Base[0];%{PE}
;FOLD Parameters ;%{h}
;Params IlfProvider=kukaroboter.basistech.inlineforms.movement.spline; Kuka.IsGlobalPoint=False; Kuka.PointName=P550; Kuka.BlendingEnabled=False; Kuka.MoveDataName=CPDAT550; Kuka.VelocityPath=1.000; Kuka.VelocityFieldEnabled=True; Kuka.ColDetectFieldEnabled=True; Kuka.CurrentCDSetIndex=0; Kuka.MovementParameterFieldEnabled=True; IlfCommand=SLIN
;ENDFOLD
SLIN XP550 WITH $VEL = SVEL_CP(2.0, , LCPDAT550),$TOOL = STOOL2(FP550),$BASE = SBASE(FP550.BASE_NO),$IPO_MODE = SIPO_MODE(FP550.IPO_FRAME),$LOAD = SLOAD(FP550.TOOL_NO),$ACC = SACC_CP(LCPDAT550),$ORI_TYPE = SORI_TYP(LCPDAT550),$APO = SAPO(LCPDAT550),$JERK = SJERK(LCPDAT550),$COLLMON_TOL_PRO[1] = USE_CM_PRO_VALUES(0)
;ENDFOLD

;FOLD SLIN P551 Vel=1 m/s CPDAT551 Tool[4]:Microflown3D Base[0];%{PE}
;FOLD Parameters ;%{h}
;Params IlfProvider=kukaroboter.basistech.inlineforms.movement.spline; Kuka.IsGlobalPoint=False; Kuka.PointName=P551; Kuka.BlendingEnabled=False; Kuka.MoveDataName=CPDAT551; Kuka.VelocityPath=1.000; Kuka.VelocityFieldEnabled=True; Kuka.ColDetectFieldEnabled=True; Kuka.CurrentCDSetIndex=0; Kuka.MovementParameterFieldEnabled=True; IlfCommand=SLIN
;ENDFOLD
SLIN XP551 WITH $VEL = SVEL_CP(2.0, , LCPDAT551),$TOOL = STOOL2(FP551),$BASE = SBASE(FP551.BASE_NO),$IPO_MODE = SIPO_MODE(FP551.IPO_FRAME),$LOAD = SLOAD(FP551.TOOL_NO),$ACC = SACC_CP(LCPDAT551),$ORI_TYPE = SORI_TYP(LCPDAT551),$APO = SAPO(LCPDAT551),$JERK = SJERK(LCPDAT551),$COLLMON_TOL_PRO[1] = USE_CM_PRO_VALUES(0)
;ENDFOLD

;FOLD SLIN P552 Vel=1 m/s CPDAT552 Tool[4]:Microflown3D Base[0];%{PE}
;FOLD Parameters ;%{h}
;Params IlfProvider=kukaroboter.basistech.inlineforms.movement.spline; Kuka.IsGlobalPoint=False; Kuka.PointName=P552; Kuka.BlendingEnabled=False; Kuka.MoveDataName=CPDAT552; Kuka.VelocityPath=1.000; Kuka.VelocityFieldEnabled=True; Kuka.ColDetectFieldEnabled=True; Kuka.CurrentCDSetIndex=0; Kuka.MovementParameterFieldEnabled=True; IlfCommand=SLIN
;ENDFOLD
SLIN XP552 WITH $VEL = SVEL_CP(2.0, , LCPDAT552),$TOOL = STOOL2(FP552),$BASE = SBASE(FP552.BASE_NO),$IPO_MODE = SIPO_MODE(FP552.IPO_FRAME),$LOAD = SLOAD(FP552.TOOL_NO),$ACC = SACC_CP(LCPDAT552),$ORI_TYPE = SORI_TYP(LCPDAT552),$APO = SAPO(LCPDAT552),$JERK = SJERK(LCPDAT552),$COLLMON_TOL_PRO[1] = USE_CM_PRO_VALUES(0)
;ENDFOLD

;FOLD SLIN P553 Vel=1 m/s CPDAT553 Tool[4]:Microflown3D Base[0];%{PE}
;FOLD Parameters ;%{h}
;Params IlfProvider=kukaroboter.basistech.inlineforms.movement.spline; Kuka.IsGlobalPoint=False; Kuka.PointName=P553; Kuka.BlendingEnabled=False; Kuka.MoveDataName=CPDAT553; Kuka.VelocityPath=1.000; Kuka.VelocityFieldEnabled=True; Kuka.ColDetectFieldEnabled=True; Kuka.CurrentCDSetIndex=0; Kuka.MovementParameterFieldEnabled=True; IlfCommand=SLIN
;ENDFOLD
SLIN XP553 WITH $VEL = SVEL_CP(2.0, , LCPDAT553),$TOOL = STOOL2(FP553),$BASE = SBASE(FP553.BASE_NO),$IPO_MODE = SIPO_MODE(FP553.IPO_FRAME),$LOAD = SLOAD(FP553.TOOL_NO),$ACC = SACC_CP(LCPDAT553),$ORI_TYPE = SORI_TYP(LCPDAT553),$APO = SAPO(LCPDAT553),$JERK = SJERK(LCPDAT553),$COLLMON_TOL_PRO[1] = USE_CM_PRO_VALUES(0)
;ENDFOLD

;FOLD SLIN P554 Vel=1 m/s CPDAT554 Tool[4]:Microflown3D Base[0];%{PE}
;FOLD Parameters ;%{h}
;Params IlfProvider=kukaroboter.basistech.inlineforms.movement.spline; Kuka.IsGlobalPoint=False; Kuka.PointName=P554; Kuka.BlendingEnabled=False; Kuka.MoveDataName=CPDAT554; Kuka.VelocityPath=1.000; Kuka.VelocityFieldEnabled=True; Kuka.ColDetectFieldEnabled=True; Kuka.CurrentCDSetIndex=0; Kuka.MovementParameterFieldEnabled=True; IlfCommand=SLIN
;ENDFOLD
SLIN XP554 WITH $VEL = SVEL_CP(2.0, , LCPDAT554),$TOOL = STOOL2(FP554),$BASE = SBASE(FP554.BASE_NO),$IPO_MODE = SIPO_MODE(FP554.IPO_FRAME),$LOAD = SLOAD(FP554.TOOL_NO),$ACC = SACC_CP(LCPDAT554),$ORI_TYPE = SORI_TYP(LCPDAT554),$APO = SAPO(LCPDAT554),$JERK = SJERK(LCPDAT554),$COLLMON_TOL_PRO[1] = USE_CM_PRO_VALUES(0)
;ENDFOLD

;FOLD SLIN P555 Vel=1 m/s CPDAT555 Tool[4]:Microflown3D Base[0];%{PE}
;FOLD Parameters ;%{h}
;Params IlfProvider=kukaroboter.basistech.inlineforms.movement.spline; Kuka.IsGlobalPoint=False; Kuka.PointName=P555; Kuka.BlendingEnabled=False; Kuka.MoveDataName=CPDAT555; Kuka.VelocityPath=1.000; Kuka.VelocityFieldEnabled=True; Kuka.ColDetectFieldEnabled=True; Kuka.CurrentCDSetIndex=0; Kuka.MovementParameterFieldEnabled=True; IlfCommand=SLIN
;ENDFOLD
SLIN XP555 WITH $VEL = SVEL_CP(2.0, , LCPDAT555),$TOOL = STOOL2(FP555),$BASE = SBASE(FP555.BASE_NO),$IPO_MODE = SIPO_MODE(FP555.IPO_FRAME),$LOAD = SLOAD(FP555.TOOL_NO),$ACC = SACC_CP(LCPDAT555),$ORI_TYPE = SORI_TYP(LCPDAT555),$APO = SAPO(LCPDAT555),$JERK = SJERK(LCPDAT555),$COLLMON_TOL_PRO[1] = USE_CM_PRO_VALUES(0)
;ENDFOLD

;FOLD SLIN P556 Vel=1 m/s CPDAT556 Tool[4]:Microflown3D Base[0];%{PE}
;FOLD Parameters ;%{h}
;Params IlfProvider=kukaroboter.basistech.inlineforms.movement.spline; Kuka.IsGlobalPoint=False; Kuka.PointName=P556; Kuka.BlendingEnabled=False; Kuka.MoveDataName=CPDAT556; Kuka.VelocityPath=1.000; Kuka.VelocityFieldEnabled=True; Kuka.ColDetectFieldEnabled=True; Kuka.CurrentCDSetIndex=0; Kuka.MovementParameterFieldEnabled=True; IlfCommand=SLIN
;ENDFOLD
SLIN XP556 WITH $VEL = SVEL_CP(2.0, , LCPDAT556),$TOOL = STOOL2(FP556),$BASE = SBASE(FP556.BASE_NO),$IPO_MODE = SIPO_MODE(FP556.IPO_FRAME),$LOAD = SLOAD(FP556.TOOL_NO),$ACC = SACC_CP(LCPDAT556),$ORI_TYPE = SORI_TYP(LCPDAT556),$APO = SAPO(LCPDAT556),$JERK = SJERK(LCPDAT556),$COLLMON_TOL_PRO[1] = USE_CM_PRO_VALUES(0)
;ENDFOLD

;FOLD SLIN P557 Vel=1 m/s CPDAT557 Tool[4]:Microflown3D Base[0];%{PE}
;FOLD Parameters ;%{h}
;Params IlfProvider=kukaroboter.basistech.inlineforms.movement.spline; Kuka.IsGlobalPoint=False; Kuka.PointName=P557; Kuka.BlendingEnabled=False; Kuka.MoveDataName=CPDAT557; Kuka.VelocityPath=1.000; Kuka.VelocityFieldEnabled=True; Kuka.ColDetectFieldEnabled=True; Kuka.CurrentCDSetIndex=0; Kuka.MovementParameterFieldEnabled=True; IlfCommand=SLIN
;ENDFOLD
SLIN XP557 WITH $VEL = SVEL_CP(2.0, , LCPDAT557),$TOOL = STOOL2(FP557),$BASE = SBASE(FP557.BASE_NO),$IPO_MODE = SIPO_MODE(FP557.IPO_FRAME),$LOAD = SLOAD(FP557.TOOL_NO),$ACC = SACC_CP(LCPDAT557),$ORI_TYPE = SORI_TYP(LCPDAT557),$APO = SAPO(LCPDAT557),$JERK = SJERK(LCPDAT557),$COLLMON_TOL_PRO[1] = USE_CM_PRO_VALUES(0)
;ENDFOLD

;FOLD SLIN P558 Vel=1 m/s CPDAT558 Tool[4]:Microflown3D Base[0];%{PE}
;FOLD Parameters ;%{h}
;Params IlfProvider=kukaroboter.basistech.inlineforms.movement.spline; Kuka.IsGlobalPoint=False; Kuka.PointName=P558; Kuka.BlendingEnabled=False; Kuka.MoveDataName=CPDAT558; Kuka.VelocityPath=1.000; Kuka.VelocityFieldEnabled=True; Kuka.ColDetectFieldEnabled=True; Kuka.CurrentCDSetIndex=0; Kuka.MovementParameterFieldEnabled=True; IlfCommand=SLIN
;ENDFOLD
SLIN XP558 WITH $VEL = SVEL_CP(2.0, , LCPDAT558),$TOOL = STOOL2(FP558),$BASE = SBASE(FP558.BASE_NO),$IPO_MODE = SIPO_MODE(FP558.IPO_FRAME),$LOAD = SLOAD(FP558.TOOL_NO),$ACC = SACC_CP(LCPDAT558),$ORI_TYPE = SORI_TYP(LCPDAT558),$APO = SAPO(LCPDAT558),$JERK = SJERK(LCPDAT558),$COLLMON_TOL_PRO[1] = USE_CM_PRO_VALUES(0)
;ENDFOLD

;FOLD SLIN P559 Vel=1 m/s CPDAT559 Tool[4]:Microflown3D Base[0];%{PE}
;FOLD Parameters ;%{h}
;Params IlfProvider=kukaroboter.basistech.inlineforms.movement.spline; Kuka.IsGlobalPoint=False; Kuka.PointName=P559; Kuka.BlendingEnabled=False; Kuka.MoveDataName=CPDAT559; Kuka.VelocityPath=1.000; Kuka.VelocityFieldEnabled=True; Kuka.ColDetectFieldEnabled=True; Kuka.CurrentCDSetIndex=0; Kuka.MovementParameterFieldEnabled=True; IlfCommand=SLIN
;ENDFOLD
SLIN XP559 WITH $VEL = SVEL_CP(2.0, , LCPDAT559),$TOOL = STOOL2(FP559),$BASE = SBASE(FP559.BASE_NO),$IPO_MODE = SIPO_MODE(FP559.IPO_FRAME),$LOAD = SLOAD(FP559.TOOL_NO),$ACC = SACC_CP(LCPDAT559),$ORI_TYPE = SORI_TYP(LCPDAT559),$APO = SAPO(LCPDAT559),$JERK = SJERK(LCPDAT559),$COLLMON_TOL_PRO[1] = USE_CM_PRO_VALUES(0)
;ENDFOLD

;FOLD SLIN P560 Vel=1 m/s CPDAT560 Tool[4]:Microflown3D Base[0];%{PE}
;FOLD Parameters ;%{h}
;Params IlfProvider=kukaroboter.basistech.inlineforms.movement.spline; Kuka.IsGlobalPoint=False; Kuka.PointName=P560; Kuka.BlendingEnabled=False; Kuka.MoveDataName=CPDAT560; Kuka.VelocityPath=1.000; Kuka.VelocityFieldEnabled=True; Kuka.ColDetectFieldEnabled=True; Kuka.CurrentCDSetIndex=0; Kuka.MovementParameterFieldEnabled=True; IlfCommand=SLIN
;ENDFOLD
SLIN XP560 WITH $VEL = SVEL_CP(2.0, , LCPDAT560),$TOOL = STOOL2(FP560),$BASE = SBASE(FP560.BASE_NO),$IPO_MODE = SIPO_MODE(FP560.IPO_FRAME),$LOAD = SLOAD(FP560.TOOL_NO),$ACC = SACC_CP(LCPDAT560),$ORI_TYPE = SORI_TYP(LCPDAT560),$APO = SAPO(LCPDAT560),$JERK = SJERK(LCPDAT560),$COLLMON_TOL_PRO[1] = USE_CM_PRO_VALUES(0)
;ENDFOLD

;FOLD SLIN P561 Vel=1 m/s CPDAT561 Tool[4]:Microflown3D Base[0];%{PE}
;FOLD Parameters ;%{h}
;Params IlfProvider=kukaroboter.basistech.inlineforms.movement.spline; Kuka.IsGlobalPoint=False; Kuka.PointName=P561; Kuka.BlendingEnabled=False; Kuka.MoveDataName=CPDAT561; Kuka.VelocityPath=1.000; Kuka.VelocityFieldEnabled=True; Kuka.ColDetectFieldEnabled=True; Kuka.CurrentCDSetIndex=0; Kuka.MovementParameterFieldEnabled=True; IlfCommand=SLIN
;ENDFOLD
SLIN XP561 WITH $VEL = SVEL_CP(2.0, , LCPDAT561),$TOOL = STOOL2(FP561),$BASE = SBASE(FP561.BASE_NO),$IPO_MODE = SIPO_MODE(FP561.IPO_FRAME),$LOAD = SLOAD(FP561.TOOL_NO),$ACC = SACC_CP(LCPDAT561),$ORI_TYPE = SORI_TYP(LCPDAT561),$APO = SAPO(LCPDAT561),$JERK = SJERK(LCPDAT561),$COLLMON_TOL_PRO[1] = USE_CM_PRO_VALUES(0)
;ENDFOLD

;FOLD SLIN P562 Vel=1 m/s CPDAT562 Tool[4]:Microflown3D Base[0];%{PE}
;FOLD Parameters ;%{h}
;Params IlfProvider=kukaroboter.basistech.inlineforms.movement.spline; Kuka.IsGlobalPoint=False; Kuka.PointName=P562; Kuka.BlendingEnabled=False; Kuka.MoveDataName=CPDAT562; Kuka.VelocityPath=1.000; Kuka.VelocityFieldEnabled=True; Kuka.ColDetectFieldEnabled=True; Kuka.CurrentCDSetIndex=0; Kuka.MovementParameterFieldEnabled=True; IlfCommand=SLIN
;ENDFOLD
SLIN XP562 WITH $VEL = SVEL_CP(2.0, , LCPDAT562),$TOOL = STOOL2(FP562),$BASE = SBASE(FP562.BASE_NO),$IPO_MODE = SIPO_MODE(FP562.IPO_FRAME),$LOAD = SLOAD(FP562.TOOL_NO),$ACC = SACC_CP(LCPDAT562),$ORI_TYPE = SORI_TYP(LCPDAT562),$APO = SAPO(LCPDAT562),$JERK = SJERK(LCPDAT562),$COLLMON_TOL_PRO[1] = USE_CM_PRO_VALUES(0)
;ENDFOLD

;FOLD SLIN P563 Vel=1 m/s CPDAT563 Tool[4]:Microflown3D Base[0];%{PE}
;FOLD Parameters ;%{h}
;Params IlfProvider=kukaroboter.basistech.inlineforms.movement.spline; Kuka.IsGlobalPoint=False; Kuka.PointName=P563; Kuka.BlendingEnabled=False; Kuka.MoveDataName=CPDAT563; Kuka.VelocityPath=1.000; Kuka.VelocityFieldEnabled=True; Kuka.ColDetectFieldEnabled=True; Kuka.CurrentCDSetIndex=0; Kuka.MovementParameterFieldEnabled=True; IlfCommand=SLIN
;ENDFOLD
SLIN XP563 WITH $VEL = SVEL_CP(2.0, , LCPDAT563),$TOOL = STOOL2(FP563),$BASE = SBASE(FP563.BASE_NO),$IPO_MODE = SIPO_MODE(FP563.IPO_FRAME),$LOAD = SLOAD(FP563.TOOL_NO),$ACC = SACC_CP(LCPDAT563),$ORI_TYPE = SORI_TYP(LCPDAT563),$APO = SAPO(LCPDAT563),$JERK = SJERK(LCPDAT563),$COLLMON_TOL_PRO[1] = USE_CM_PRO_VALUES(0)
;ENDFOLD

;FOLD SLIN P564 Vel=1 m/s CPDAT564 Tool[4]:Microflown3D Base[0];%{PE}
;FOLD Parameters ;%{h}
;Params IlfProvider=kukaroboter.basistech.inlineforms.movement.spline; Kuka.IsGlobalPoint=False; Kuka.PointName=P564; Kuka.BlendingEnabled=False; Kuka.MoveDataName=CPDAT564; Kuka.VelocityPath=1.000; Kuka.VelocityFieldEnabled=True; Kuka.ColDetectFieldEnabled=True; Kuka.CurrentCDSetIndex=0; Kuka.MovementParameterFieldEnabled=True; IlfCommand=SLIN
;ENDFOLD
SLIN XP564 WITH $VEL = SVEL_CP(2.0, , LCPDAT564),$TOOL = STOOL2(FP564),$BASE = SBASE(FP564.BASE_NO),$IPO_MODE = SIPO_MODE(FP564.IPO_FRAME),$LOAD = SLOAD(FP564.TOOL_NO),$ACC = SACC_CP(LCPDAT564),$ORI_TYPE = SORI_TYP(LCPDAT564),$APO = SAPO(LCPDAT564),$JERK = SJERK(LCPDAT564),$COLLMON_TOL_PRO[1] = USE_CM_PRO_VALUES(0)
;ENDFOLD

;FOLD SLIN P565 Vel=1 m/s CPDAT565 Tool[4]:Microflown3D Base[0];%{PE}
;FOLD Parameters ;%{h}
;Params IlfProvider=kukaroboter.basistech.inlineforms.movement.spline; Kuka.IsGlobalPoint=False; Kuka.PointName=P565; Kuka.BlendingEnabled=False; Kuka.MoveDataName=CPDAT565; Kuka.VelocityPath=1.000; Kuka.VelocityFieldEnabled=True; Kuka.ColDetectFieldEnabled=True; Kuka.CurrentCDSetIndex=0; Kuka.MovementParameterFieldEnabled=True; IlfCommand=SLIN
;ENDFOLD
SLIN XP565 WITH $VEL = SVEL_CP(2.0, , LCPDAT565),$TOOL = STOOL2(FP565),$BASE = SBASE(FP565.BASE_NO),$IPO_MODE = SIPO_MODE(FP565.IPO_FRAME),$LOAD = SLOAD(FP565.TOOL_NO),$ACC = SACC_CP(LCPDAT565),$ORI_TYPE = SORI_TYP(LCPDAT565),$APO = SAPO(LCPDAT565),$JERK = SJERK(LCPDAT565),$COLLMON_TOL_PRO[1] = USE_CM_PRO_VALUES(0)
;ENDFOLD

;FOLD SLIN P566 Vel=1 m/s CPDAT566 Tool[4]:Microflown3D Base[0];%{PE}
;FOLD Parameters ;%{h}
;Params IlfProvider=kukaroboter.basistech.inlineforms.movement.spline; Kuka.IsGlobalPoint=False; Kuka.PointName=P566; Kuka.BlendingEnabled=False; Kuka.MoveDataName=CPDAT566; Kuka.VelocityPath=1.000; Kuka.VelocityFieldEnabled=True; Kuka.ColDetectFieldEnabled=True; Kuka.CurrentCDSetIndex=0; Kuka.MovementParameterFieldEnabled=True; IlfCommand=SLIN
;ENDFOLD
SLIN XP566 WITH $VEL = SVEL_CP(2.0, , LCPDAT566),$TOOL = STOOL2(FP566),$BASE = SBASE(FP566.BASE_NO),$IPO_MODE = SIPO_MODE(FP566.IPO_FRAME),$LOAD = SLOAD(FP566.TOOL_NO),$ACC = SACC_CP(LCPDAT566),$ORI_TYPE = SORI_TYP(LCPDAT566),$APO = SAPO(LCPDAT566),$JERK = SJERK(LCPDAT566),$COLLMON_TOL_PRO[1] = USE_CM_PRO_VALUES(0)
;ENDFOLD

;FOLD SLIN P567 Vel=1 m/s CPDAT567 Tool[4]:Microflown3D Base[0];%{PE}
;FOLD Parameters ;%{h}
;Params IlfProvider=kukaroboter.basistech.inlineforms.movement.spline; Kuka.IsGlobalPoint=False; Kuka.PointName=P567; Kuka.BlendingEnabled=False; Kuka.MoveDataName=CPDAT567; Kuka.VelocityPath=1.000; Kuka.VelocityFieldEnabled=True; Kuka.ColDetectFieldEnabled=True; Kuka.CurrentCDSetIndex=0; Kuka.MovementParameterFieldEnabled=True; IlfCommand=SLIN
;ENDFOLD
SLIN XP567 WITH $VEL = SVEL_CP(2.0, , LCPDAT567),$TOOL = STOOL2(FP567),$BASE = SBASE(FP567.BASE_NO),$IPO_MODE = SIPO_MODE(FP567.IPO_FRAME),$LOAD = SLOAD(FP567.TOOL_NO),$ACC = SACC_CP(LCPDAT567),$ORI_TYPE = SORI_TYP(LCPDAT567),$APO = SAPO(LCPDAT567),$JERK = SJERK(LCPDAT567),$COLLMON_TOL_PRO[1] = USE_CM_PRO_VALUES(0)
;ENDFOLD

;FOLD SLIN P568 Vel=1 m/s CPDAT568 Tool[4]:Microflown3D Base[0];%{PE}
;FOLD Parameters ;%{h}
;Params IlfProvider=kukaroboter.basistech.inlineforms.movement.spline; Kuka.IsGlobalPoint=False; Kuka.PointName=P568; Kuka.BlendingEnabled=False; Kuka.MoveDataName=CPDAT568; Kuka.VelocityPath=1.000; Kuka.VelocityFieldEnabled=True; Kuka.ColDetectFieldEnabled=True; Kuka.CurrentCDSetIndex=0; Kuka.MovementParameterFieldEnabled=True; IlfCommand=SLIN
;ENDFOLD
SLIN XP568 WITH $VEL = SVEL_CP(2.0, , LCPDAT568),$TOOL = STOOL2(FP568),$BASE = SBASE(FP568.BASE_NO),$IPO_MODE = SIPO_MODE(FP568.IPO_FRAME),$LOAD = SLOAD(FP568.TOOL_NO),$ACC = SACC_CP(LCPDAT568),$ORI_TYPE = SORI_TYP(LCPDAT568),$APO = SAPO(LCPDAT568),$JERK = SJERK(LCPDAT568),$COLLMON_TOL_PRO[1] = USE_CM_PRO_VALUES(0)
;ENDFOLD

;FOLD SLIN P569 Vel=1 m/s CPDAT569 Tool[4]:Microflown3D Base[0];%{PE}
;FOLD Parameters ;%{h}
;Params IlfProvider=kukaroboter.basistech.inlineforms.movement.spline; Kuka.IsGlobalPoint=False; Kuka.PointName=P569; Kuka.BlendingEnabled=False; Kuka.MoveDataName=CPDAT569; Kuka.VelocityPath=1.000; Kuka.VelocityFieldEnabled=True; Kuka.ColDetectFieldEnabled=True; Kuka.CurrentCDSetIndex=0; Kuka.MovementParameterFieldEnabled=True; IlfCommand=SLIN
;ENDFOLD
SLIN XP569 WITH $VEL = SVEL_CP(2.0, , LCPDAT569),$TOOL = STOOL2(FP569),$BASE = SBASE(FP569.BASE_NO),$IPO_MODE = SIPO_MODE(FP569.IPO_FRAME),$LOAD = SLOAD(FP569.TOOL_NO),$ACC = SACC_CP(LCPDAT569),$ORI_TYPE = SORI_TYP(LCPDAT569),$APO = SAPO(LCPDAT569),$JERK = SJERK(LCPDAT569),$COLLMON_TOL_PRO[1] = USE_CM_PRO_VALUES(0)
;ENDFOLD

;FOLD SLIN P570 Vel=1 m/s CPDAT570 Tool[4]:Microflown3D Base[0];%{PE}
;FOLD Parameters ;%{h}
;Params IlfProvider=kukaroboter.basistech.inlineforms.movement.spline; Kuka.IsGlobalPoint=False; Kuka.PointName=P570; Kuka.BlendingEnabled=False; Kuka.MoveDataName=CPDAT570; Kuka.VelocityPath=1.000; Kuka.VelocityFieldEnabled=True; Kuka.ColDetectFieldEnabled=True; Kuka.CurrentCDSetIndex=0; Kuka.MovementParameterFieldEnabled=True; IlfCommand=SLIN
;ENDFOLD
SLIN XP570 WITH $VEL = SVEL_CP(2.0, , LCPDAT570),$TOOL = STOOL2(FP570),$BASE = SBASE(FP570.BASE_NO),$IPO_MODE = SIPO_MODE(FP570.IPO_FRAME),$LOAD = SLOAD(FP570.TOOL_NO),$ACC = SACC_CP(LCPDAT570),$ORI_TYPE = SORI_TYP(LCPDAT570),$APO = SAPO(LCPDAT570),$JERK = SJERK(LCPDAT570),$COLLMON_TOL_PRO[1] = USE_CM_PRO_VALUES(0)
;ENDFOLD

;FOLD SLIN P571 Vel=1 m/s CPDAT571 Tool[4]:Microflown3D Base[0];%{PE}
;FOLD Parameters ;%{h}
;Params IlfProvider=kukaroboter.basistech.inlineforms.movement.spline; Kuka.IsGlobalPoint=False; Kuka.PointName=P571; Kuka.BlendingEnabled=False; Kuka.MoveDataName=CPDAT571; Kuka.VelocityPath=1.000; Kuka.VelocityFieldEnabled=True; Kuka.ColDetectFieldEnabled=True; Kuka.CurrentCDSetIndex=0; Kuka.MovementParameterFieldEnabled=True; IlfCommand=SLIN
;ENDFOLD
SLIN XP571 WITH $VEL = SVEL_CP(2.0, , LCPDAT571),$TOOL = STOOL2(FP571),$BASE = SBASE(FP571.BASE_NO),$IPO_MODE = SIPO_MODE(FP571.IPO_FRAME),$LOAD = SLOAD(FP571.TOOL_NO),$ACC = SACC_CP(LCPDAT571),$ORI_TYPE = SORI_TYP(LCPDAT571),$APO = SAPO(LCPDAT571),$JERK = SJERK(LCPDAT571),$COLLMON_TOL_PRO[1] = USE_CM_PRO_VALUES(0)
;ENDFOLD

;FOLD SLIN P572 Vel=1 m/s CPDAT572 Tool[4]:Microflown3D Base[0];%{PE}
;FOLD Parameters ;%{h}
;Params IlfProvider=kukaroboter.basistech.inlineforms.movement.spline; Kuka.IsGlobalPoint=False; Kuka.PointName=P572; Kuka.BlendingEnabled=False; Kuka.MoveDataName=CPDAT572; Kuka.VelocityPath=1.000; Kuka.VelocityFieldEnabled=True; Kuka.ColDetectFieldEnabled=True; Kuka.CurrentCDSetIndex=0; Kuka.MovementParameterFieldEnabled=True; IlfCommand=SLIN
;ENDFOLD
SLIN XP572 WITH $VEL = SVEL_CP(2.0, , LCPDAT572),$TOOL = STOOL2(FP572),$BASE = SBASE(FP572.BASE_NO),$IPO_MODE = SIPO_MODE(FP572.IPO_FRAME),$LOAD = SLOAD(FP572.TOOL_NO),$ACC = SACC_CP(LCPDAT572),$ORI_TYPE = SORI_TYP(LCPDAT572),$APO = SAPO(LCPDAT572),$JERK = SJERK(LCPDAT572),$COLLMON_TOL_PRO[1] = USE_CM_PRO_VALUES(0)
;ENDFOLD

;FOLD SLIN P573 Vel=1 m/s CPDAT573 Tool[4]:Microflown3D Base[0];%{PE}
;FOLD Parameters ;%{h}
;Params IlfProvider=kukaroboter.basistech.inlineforms.movement.spline; Kuka.IsGlobalPoint=False; Kuka.PointName=P573; Kuka.BlendingEnabled=False; Kuka.MoveDataName=CPDAT573; Kuka.VelocityPath=1.000; Kuka.VelocityFieldEnabled=True; Kuka.ColDetectFieldEnabled=True; Kuka.CurrentCDSetIndex=0; Kuka.MovementParameterFieldEnabled=True; IlfCommand=SLIN
;ENDFOLD
SLIN XP573 WITH $VEL = SVEL_CP(2.0, , LCPDAT573),$TOOL = STOOL2(FP573),$BASE = SBASE(FP573.BASE_NO),$IPO_MODE = SIPO_MODE(FP573.IPO_FRAME),$LOAD = SLOAD(FP573.TOOL_NO),$ACC = SACC_CP(LCPDAT573),$ORI_TYPE = SORI_TYP(LCPDAT573),$APO = SAPO(LCPDAT573),$JERK = SJERK(LCPDAT573),$COLLMON_TOL_PRO[1] = USE_CM_PRO_VALUES(0)
;ENDFOLD

;FOLD SLIN P574 Vel=1 m/s CPDAT574 Tool[4]:Microflown3D Base[0];%{PE}
;FOLD Parameters ;%{h}
;Params IlfProvider=kukaroboter.basistech.inlineforms.movement.spline; Kuka.IsGlobalPoint=False; Kuka.PointName=P574; Kuka.BlendingEnabled=False; Kuka.MoveDataName=CPDAT574; Kuka.VelocityPath=1.000; Kuka.VelocityFieldEnabled=True; Kuka.ColDetectFieldEnabled=True; Kuka.CurrentCDSetIndex=0; Kuka.MovementParameterFieldEnabled=True; IlfCommand=SLIN
;ENDFOLD
SLIN XP574 WITH $VEL = SVEL_CP(2.0, , LCPDAT574),$TOOL = STOOL2(FP574),$BASE = SBASE(FP574.BASE_NO),$IPO_MODE = SIPO_MODE(FP574.IPO_FRAME),$LOAD = SLOAD(FP574.TOOL_NO),$ACC = SACC_CP(LCPDAT574),$ORI_TYPE = SORI_TYP(LCPDAT574),$APO = SAPO(LCPDAT574),$JERK = SJERK(LCPDAT574),$COLLMON_TOL_PRO[1] = USE_CM_PRO_VALUES(0)
;ENDFOLD

;FOLD SLIN P575 Vel=1 m/s CPDAT575 Tool[4]:Microflown3D Base[0];%{PE}
;FOLD Parameters ;%{h}
;Params IlfProvider=kukaroboter.basistech.inlineforms.movement.spline; Kuka.IsGlobalPoint=False; Kuka.PointName=P575; Kuka.BlendingEnabled=False; Kuka.MoveDataName=CPDAT575; Kuka.VelocityPath=1.000; Kuka.VelocityFieldEnabled=True; Kuka.ColDetectFieldEnabled=True; Kuka.CurrentCDSetIndex=0; Kuka.MovementParameterFieldEnabled=True; IlfCommand=SLIN
;ENDFOLD
SLIN XP575 WITH $VEL = SVEL_CP(2.0, , LCPDAT575),$TOOL = STOOL2(FP575),$BASE = SBASE(FP575.BASE_NO),$IPO_MODE = SIPO_MODE(FP575.IPO_FRAME),$LOAD = SLOAD(FP575.TOOL_NO),$ACC = SACC_CP(LCPDAT575),$ORI_TYPE = SORI_TYP(LCPDAT575),$APO = SAPO(LCPDAT575),$JERK = SJERK(LCPDAT575),$COLLMON_TOL_PRO[1] = USE_CM_PRO_VALUES(0)
;ENDFOLD

;FOLD SLIN P576 Vel=1 m/s CPDAT576 Tool[4]:Microflown3D Base[0];%{PE}
;FOLD Parameters ;%{h}
;Params IlfProvider=kukaroboter.basistech.inlineforms.movement.spline; Kuka.IsGlobalPoint=False; Kuka.PointName=P576; Kuka.BlendingEnabled=False; Kuka.MoveDataName=CPDAT576; Kuka.VelocityPath=1.000; Kuka.VelocityFieldEnabled=True; Kuka.ColDetectFieldEnabled=True; Kuka.CurrentCDSetIndex=0; Kuka.MovementParameterFieldEnabled=True; IlfCommand=SLIN
;ENDFOLD
SLIN XP576 WITH $VEL = SVEL_CP(2.0, , LCPDAT576),$TOOL = STOOL2(FP576),$BASE = SBASE(FP576.BASE_NO),$IPO_MODE = SIPO_MODE(FP576.IPO_FRAME),$LOAD = SLOAD(FP576.TOOL_NO),$ACC = SACC_CP(LCPDAT576),$ORI_TYPE = SORI_TYP(LCPDAT576),$APO = SAPO(LCPDAT576),$JERK = SJERK(LCPDAT576),$COLLMON_TOL_PRO[1] = USE_CM_PRO_VALUES(0)
;ENDFOLD

;FOLD SLIN P577 Vel=1 m/s CPDAT577 Tool[4]:Microflown3D Base[0];%{PE}
;FOLD Parameters ;%{h}
;Params IlfProvider=kukaroboter.basistech.inlineforms.movement.spline; Kuka.IsGlobalPoint=False; Kuka.PointName=P577; Kuka.BlendingEnabled=False; Kuka.MoveDataName=CPDAT577; Kuka.VelocityPath=1.000; Kuka.VelocityFieldEnabled=True; Kuka.ColDetectFieldEnabled=True; Kuka.CurrentCDSetIndex=0; Kuka.MovementParameterFieldEnabled=True; IlfCommand=SLIN
;ENDFOLD
SLIN XP577 WITH $VEL = SVEL_CP(2.0, , LCPDAT577),$TOOL = STOOL2(FP577),$BASE = SBASE(FP577.BASE_NO),$IPO_MODE = SIPO_MODE(FP577.IPO_FRAME),$LOAD = SLOAD(FP577.TOOL_NO),$ACC = SACC_CP(LCPDAT577),$ORI_TYPE = SORI_TYP(LCPDAT577),$APO = SAPO(LCPDAT577),$JERK = SJERK(LCPDAT577),$COLLMON_TOL_PRO[1] = USE_CM_PRO_VALUES(0)
;ENDFOLD

;FOLD SLIN P578 Vel=1 m/s CPDAT578 Tool[4]:Microflown3D Base[0];%{PE}
;FOLD Parameters ;%{h}
;Params IlfProvider=kukaroboter.basistech.inlineforms.movement.spline; Kuka.IsGlobalPoint=False; Kuka.PointName=P578; Kuka.BlendingEnabled=False; Kuka.MoveDataName=CPDAT578; Kuka.VelocityPath=1.000; Kuka.VelocityFieldEnabled=True; Kuka.ColDetectFieldEnabled=True; Kuka.CurrentCDSetIndex=0; Kuka.MovementParameterFieldEnabled=True; IlfCommand=SLIN
;ENDFOLD
SLIN XP578 WITH $VEL = SVEL_CP(2.0, , LCPDAT578),$TOOL = STOOL2(FP578),$BASE = SBASE(FP578.BASE_NO),$IPO_MODE = SIPO_MODE(FP578.IPO_FRAME),$LOAD = SLOAD(FP578.TOOL_NO),$ACC = SACC_CP(LCPDAT578),$ORI_TYPE = SORI_TYP(LCPDAT578),$APO = SAPO(LCPDAT578),$JERK = SJERK(LCPDAT578),$COLLMON_TOL_PRO[1] = USE_CM_PRO_VALUES(0)
;ENDFOLD

;FOLD SLIN P579 Vel=1 m/s CPDAT579 Tool[4]:Microflown3D Base[0];%{PE}
;FOLD Parameters ;%{h}
;Params IlfProvider=kukaroboter.basistech.inlineforms.movement.spline; Kuka.IsGlobalPoint=False; Kuka.PointName=P579; Kuka.BlendingEnabled=False; Kuka.MoveDataName=CPDAT579; Kuka.VelocityPath=1.000; Kuka.VelocityFieldEnabled=True; Kuka.ColDetectFieldEnabled=True; Kuka.CurrentCDSetIndex=0; Kuka.MovementParameterFieldEnabled=True; IlfCommand=SLIN
;ENDFOLD
SLIN XP579 WITH $VEL = SVEL_CP(2.0, , LCPDAT579),$TOOL = STOOL2(FP579),$BASE = SBASE(FP579.BASE_NO),$IPO_MODE = SIPO_MODE(FP579.IPO_FRAME),$LOAD = SLOAD(FP579.TOOL_NO),$ACC = SACC_CP(LCPDAT579),$ORI_TYPE = SORI_TYP(LCPDAT579),$APO = SAPO(LCPDAT579),$JERK = SJERK(LCPDAT579),$COLLMON_TOL_PRO[1] = USE_CM_PRO_VALUES(0)
;ENDFOLD

;FOLD SLIN P580 Vel=1 m/s CPDAT580 Tool[4]:Microflown3D Base[0];%{PE}
;FOLD Parameters ;%{h}
;Params IlfProvider=kukaroboter.basistech.inlineforms.movement.spline; Kuka.IsGlobalPoint=False; Kuka.PointName=P580; Kuka.BlendingEnabled=False; Kuka.MoveDataName=CPDAT580; Kuka.VelocityPath=1.000; Kuka.VelocityFieldEnabled=True; Kuka.ColDetectFieldEnabled=True; Kuka.CurrentCDSetIndex=0; Kuka.MovementParameterFieldEnabled=True; IlfCommand=SLIN
;ENDFOLD
SLIN XP580 WITH $VEL = SVEL_CP(2.0, , LCPDAT580),$TOOL = STOOL2(FP580),$BASE = SBASE(FP580.BASE_NO),$IPO_MODE = SIPO_MODE(FP580.IPO_FRAME),$LOAD = SLOAD(FP580.TOOL_NO),$ACC = SACC_CP(LCPDAT580),$ORI_TYPE = SORI_TYP(LCPDAT580),$APO = SAPO(LCPDAT580),$JERK = SJERK(LCPDAT580),$COLLMON_TOL_PRO[1] = USE_CM_PRO_VALUES(0)
;ENDFOLD

;FOLD SLIN P581 Vel=1 m/s CPDAT581 Tool[4]:Microflown3D Base[0];%{PE}
;FOLD Parameters ;%{h}
;Params IlfProvider=kukaroboter.basistech.inlineforms.movement.spline; Kuka.IsGlobalPoint=False; Kuka.PointName=P581; Kuka.BlendingEnabled=False; Kuka.MoveDataName=CPDAT581; Kuka.VelocityPath=1.000; Kuka.VelocityFieldEnabled=True; Kuka.ColDetectFieldEnabled=True; Kuka.CurrentCDSetIndex=0; Kuka.MovementParameterFieldEnabled=True; IlfCommand=SLIN
;ENDFOLD
SLIN XP581 WITH $VEL = SVEL_CP(2.0, , LCPDAT581),$TOOL = STOOL2(FP581),$BASE = SBASE(FP581.BASE_NO),$IPO_MODE = SIPO_MODE(FP581.IPO_FRAME),$LOAD = SLOAD(FP581.TOOL_NO),$ACC = SACC_CP(LCPDAT581),$ORI_TYPE = SORI_TYP(LCPDAT581),$APO = SAPO(LCPDAT581),$JERK = SJERK(LCPDAT581),$COLLMON_TOL_PRO[1] = USE_CM_PRO_VALUES(0)
;ENDFOLD

;FOLD SLIN P582 Vel=1 m/s CPDAT582 Tool[4]:Microflown3D Base[0];%{PE}
;FOLD Parameters ;%{h}
;Params IlfProvider=kukaroboter.basistech.inlineforms.movement.spline; Kuka.IsGlobalPoint=False; Kuka.PointName=P582; Kuka.BlendingEnabled=False; Kuka.MoveDataName=CPDAT582; Kuka.VelocityPath=1.000; Kuka.VelocityFieldEnabled=True; Kuka.ColDetectFieldEnabled=True; Kuka.CurrentCDSetIndex=0; Kuka.MovementParameterFieldEnabled=True; IlfCommand=SLIN
;ENDFOLD
SLIN XP582 WITH $VEL = SVEL_CP(2.0, , LCPDAT582),$TOOL = STOOL2(FP582),$BASE = SBASE(FP582.BASE_NO),$IPO_MODE = SIPO_MODE(FP582.IPO_FRAME),$LOAD = SLOAD(FP582.TOOL_NO),$ACC = SACC_CP(LCPDAT582),$ORI_TYPE = SORI_TYP(LCPDAT582),$APO = SAPO(LCPDAT582),$JERK = SJERK(LCPDAT582),$COLLMON_TOL_PRO[1] = USE_CM_PRO_VALUES(0)
;ENDFOLD

;FOLD SLIN P583 Vel=1 m/s CPDAT583 Tool[4]:Microflown3D Base[0];%{PE}
;FOLD Parameters ;%{h}
;Params IlfProvider=kukaroboter.basistech.inlineforms.movement.spline; Kuka.IsGlobalPoint=False; Kuka.PointName=P583; Kuka.BlendingEnabled=False; Kuka.MoveDataName=CPDAT583; Kuka.VelocityPath=1.000; Kuka.VelocityFieldEnabled=True; Kuka.ColDetectFieldEnabled=True; Kuka.CurrentCDSetIndex=0; Kuka.MovementParameterFieldEnabled=True; IlfCommand=SLIN
;ENDFOLD
SLIN XP583 WITH $VEL = SVEL_CP(2.0, , LCPDAT583),$TOOL = STOOL2(FP583),$BASE = SBASE(FP583.BASE_NO),$IPO_MODE = SIPO_MODE(FP583.IPO_FRAME),$LOAD = SLOAD(FP583.TOOL_NO),$ACC = SACC_CP(LCPDAT583),$ORI_TYPE = SORI_TYP(LCPDAT583),$APO = SAPO(LCPDAT583),$JERK = SJERK(LCPDAT583),$COLLMON_TOL_PRO[1] = USE_CM_PRO_VALUES(0)
;ENDFOLD

;FOLD SLIN P584 Vel=1 m/s CPDAT584 Tool[4]:Microflown3D Base[0];%{PE}
;FOLD Parameters ;%{h}
;Params IlfProvider=kukaroboter.basistech.inlineforms.movement.spline; Kuka.IsGlobalPoint=False; Kuka.PointName=P584; Kuka.BlendingEnabled=False; Kuka.MoveDataName=CPDAT584; Kuka.VelocityPath=1.000; Kuka.VelocityFieldEnabled=True; Kuka.ColDetectFieldEnabled=True; Kuka.CurrentCDSetIndex=0; Kuka.MovementParameterFieldEnabled=True; IlfCommand=SLIN
;ENDFOLD
SLIN XP584 WITH $VEL = SVEL_CP(2.0, , LCPDAT584),$TOOL = STOOL2(FP584),$BASE = SBASE(FP584.BASE_NO),$IPO_MODE = SIPO_MODE(FP584.IPO_FRAME),$LOAD = SLOAD(FP584.TOOL_NO),$ACC = SACC_CP(LCPDAT584),$ORI_TYPE = SORI_TYP(LCPDAT584),$APO = SAPO(LCPDAT584),$JERK = SJERK(LCPDAT584),$COLLMON_TOL_PRO[1] = USE_CM_PRO_VALUES(0)
;ENDFOLD

;FOLD SLIN P585 Vel=1 m/s CPDAT585 Tool[4]:Microflown3D Base[0];%{PE}
;FOLD Parameters ;%{h}
;Params IlfProvider=kukaroboter.basistech.inlineforms.movement.spline; Kuka.IsGlobalPoint=False; Kuka.PointName=P585; Kuka.BlendingEnabled=False; Kuka.MoveDataName=CPDAT585; Kuka.VelocityPath=1.000; Kuka.VelocityFieldEnabled=True; Kuka.ColDetectFieldEnabled=True; Kuka.CurrentCDSetIndex=0; Kuka.MovementParameterFieldEnabled=True; IlfCommand=SLIN
;ENDFOLD
SLIN XP585 WITH $VEL = SVEL_CP(2.0, , LCPDAT585),$TOOL = STOOL2(FP585),$BASE = SBASE(FP585.BASE_NO),$IPO_MODE = SIPO_MODE(FP585.IPO_FRAME),$LOAD = SLOAD(FP585.TOOL_NO),$ACC = SACC_CP(LCPDAT585),$ORI_TYPE = SORI_TYP(LCPDAT585),$APO = SAPO(LCPDAT585),$JERK = SJERK(LCPDAT585),$COLLMON_TOL_PRO[1] = USE_CM_PRO_VALUES(0)
;ENDFOLD

;FOLD SLIN P586 Vel=1 m/s CPDAT586 Tool[4]:Microflown3D Base[0];%{PE}
;FOLD Parameters ;%{h}
;Params IlfProvider=kukaroboter.basistech.inlineforms.movement.spline; Kuka.IsGlobalPoint=False; Kuka.PointName=P586; Kuka.BlendingEnabled=False; Kuka.MoveDataName=CPDAT586; Kuka.VelocityPath=1.000; Kuka.VelocityFieldEnabled=True; Kuka.ColDetectFieldEnabled=True; Kuka.CurrentCDSetIndex=0; Kuka.MovementParameterFieldEnabled=True; IlfCommand=SLIN
;ENDFOLD
SLIN XP586 WITH $VEL = SVEL_CP(2.0, , LCPDAT586),$TOOL = STOOL2(FP586),$BASE = SBASE(FP586.BASE_NO),$IPO_MODE = SIPO_MODE(FP586.IPO_FRAME),$LOAD = SLOAD(FP586.TOOL_NO),$ACC = SACC_CP(LCPDAT586),$ORI_TYPE = SORI_TYP(LCPDAT586),$APO = SAPO(LCPDAT586),$JERK = SJERK(LCPDAT586),$COLLMON_TOL_PRO[1] = USE_CM_PRO_VALUES(0)
;ENDFOLD

;FOLD SLIN P587 Vel=1 m/s CPDAT587 Tool[4]:Microflown3D Base[0];%{PE}
;FOLD Parameters ;%{h}
;Params IlfProvider=kukaroboter.basistech.inlineforms.movement.spline; Kuka.IsGlobalPoint=False; Kuka.PointName=P587; Kuka.BlendingEnabled=False; Kuka.MoveDataName=CPDAT587; Kuka.VelocityPath=1.000; Kuka.VelocityFieldEnabled=True; Kuka.ColDetectFieldEnabled=True; Kuka.CurrentCDSetIndex=0; Kuka.MovementParameterFieldEnabled=True; IlfCommand=SLIN
;ENDFOLD
SLIN XP587 WITH $VEL = SVEL_CP(2.0, , LCPDAT587),$TOOL = STOOL2(FP587),$BASE = SBASE(FP587.BASE_NO),$IPO_MODE = SIPO_MODE(FP587.IPO_FRAME),$LOAD = SLOAD(FP587.TOOL_NO),$ACC = SACC_CP(LCPDAT587),$ORI_TYPE = SORI_TYP(LCPDAT587),$APO = SAPO(LCPDAT587),$JERK = SJERK(LCPDAT587),$COLLMON_TOL_PRO[1] = USE_CM_PRO_VALUES(0)
;ENDFOLD

;FOLD SLIN P588 Vel=1 m/s CPDAT588 Tool[4]:Microflown3D Base[0];%{PE}
;FOLD Parameters ;%{h}
;Params IlfProvider=kukaroboter.basistech.inlineforms.movement.spline; Kuka.IsGlobalPoint=False; Kuka.PointName=P588; Kuka.BlendingEnabled=False; Kuka.MoveDataName=CPDAT588; Kuka.VelocityPath=1.000; Kuka.VelocityFieldEnabled=True; Kuka.ColDetectFieldEnabled=True; Kuka.CurrentCDSetIndex=0; Kuka.MovementParameterFieldEnabled=True; IlfCommand=SLIN
;ENDFOLD
SLIN XP588 WITH $VEL = SVEL_CP(2.0, , LCPDAT588),$TOOL = STOOL2(FP588),$BASE = SBASE(FP588.BASE_NO),$IPO_MODE = SIPO_MODE(FP588.IPO_FRAME),$LOAD = SLOAD(FP588.TOOL_NO),$ACC = SACC_CP(LCPDAT588),$ORI_TYPE = SORI_TYP(LCPDAT588),$APO = SAPO(LCPDAT588),$JERK = SJERK(LCPDAT588),$COLLMON_TOL_PRO[1] = USE_CM_PRO_VALUES(0)
;ENDFOLD

;FOLD SLIN P589 Vel=1 m/s CPDAT589 Tool[4]:Microflown3D Base[0];%{PE}
;FOLD Parameters ;%{h}
;Params IlfProvider=kukaroboter.basistech.inlineforms.movement.spline; Kuka.IsGlobalPoint=False; Kuka.PointName=P589; Kuka.BlendingEnabled=False; Kuka.MoveDataName=CPDAT589; Kuka.VelocityPath=1.000; Kuka.VelocityFieldEnabled=True; Kuka.ColDetectFieldEnabled=True; Kuka.CurrentCDSetIndex=0; Kuka.MovementParameterFieldEnabled=True; IlfCommand=SLIN
;ENDFOLD
SLIN XP589 WITH $VEL = SVEL_CP(2.0, , LCPDAT589),$TOOL = STOOL2(FP589),$BASE = SBASE(FP589.BASE_NO),$IPO_MODE = SIPO_MODE(FP589.IPO_FRAME),$LOAD = SLOAD(FP589.TOOL_NO),$ACC = SACC_CP(LCPDAT589),$ORI_TYPE = SORI_TYP(LCPDAT589),$APO = SAPO(LCPDAT589),$JERK = SJERK(LCPDAT589),$COLLMON_TOL_PRO[1] = USE_CM_PRO_VALUES(0)
;ENDFOLD

;FOLD SLIN P590 Vel=1 m/s CPDAT590 Tool[4]:Microflown3D Base[0];%{PE}
;FOLD Parameters ;%{h}
;Params IlfProvider=kukaroboter.basistech.inlineforms.movement.spline; Kuka.IsGlobalPoint=False; Kuka.PointName=P590; Kuka.BlendingEnabled=False; Kuka.MoveDataName=CPDAT590; Kuka.VelocityPath=1.000; Kuka.VelocityFieldEnabled=True; Kuka.ColDetectFieldEnabled=True; Kuka.CurrentCDSetIndex=0; Kuka.MovementParameterFieldEnabled=True; IlfCommand=SLIN
;ENDFOLD
SLIN XP590 WITH $VEL = SVEL_CP(2.0, , LCPDAT590),$TOOL = STOOL2(FP590),$BASE = SBASE(FP590.BASE_NO),$IPO_MODE = SIPO_MODE(FP590.IPO_FRAME),$LOAD = SLOAD(FP590.TOOL_NO),$ACC = SACC_CP(LCPDAT590),$ORI_TYPE = SORI_TYP(LCPDAT590),$APO = SAPO(LCPDAT590),$JERK = SJERK(LCPDAT590),$COLLMON_TOL_PRO[1] = USE_CM_PRO_VALUES(0)
;ENDFOLD

;FOLD SLIN P591 Vel=1 m/s CPDAT591 Tool[4]:Microflown3D Base[0];%{PE}
;FOLD Parameters ;%{h}
;Params IlfProvider=kukaroboter.basistech.inlineforms.movement.spline; Kuka.IsGlobalPoint=False; Kuka.PointName=P591; Kuka.BlendingEnabled=False; Kuka.MoveDataName=CPDAT591; Kuka.VelocityPath=1.000; Kuka.VelocityFieldEnabled=True; Kuka.ColDetectFieldEnabled=True; Kuka.CurrentCDSetIndex=0; Kuka.MovementParameterFieldEnabled=True; IlfCommand=SLIN
;ENDFOLD
SLIN XP591 WITH $VEL = SVEL_CP(2.0, , LCPDAT591),$TOOL = STOOL2(FP591),$BASE = SBASE(FP591.BASE_NO),$IPO_MODE = SIPO_MODE(FP591.IPO_FRAME),$LOAD = SLOAD(FP591.TOOL_NO),$ACC = SACC_CP(LCPDAT591),$ORI_TYPE = SORI_TYP(LCPDAT591),$APO = SAPO(LCPDAT591),$JERK = SJERK(LCPDAT591),$COLLMON_TOL_PRO[1] = USE_CM_PRO_VALUES(0)
;ENDFOLD

;FOLD SLIN P592 Vel=1 m/s CPDAT592 Tool[4]:Microflown3D Base[0];%{PE}
;FOLD Parameters ;%{h}
;Params IlfProvider=kukaroboter.basistech.inlineforms.movement.spline; Kuka.IsGlobalPoint=False; Kuka.PointName=P592; Kuka.BlendingEnabled=False; Kuka.MoveDataName=CPDAT592; Kuka.VelocityPath=1.000; Kuka.VelocityFieldEnabled=True; Kuka.ColDetectFieldEnabled=True; Kuka.CurrentCDSetIndex=0; Kuka.MovementParameterFieldEnabled=True; IlfCommand=SLIN
;ENDFOLD
SLIN XP592 WITH $VEL = SVEL_CP(2.0, , LCPDAT592),$TOOL = STOOL2(FP592),$BASE = SBASE(FP592.BASE_NO),$IPO_MODE = SIPO_MODE(FP592.IPO_FRAME),$LOAD = SLOAD(FP592.TOOL_NO),$ACC = SACC_CP(LCPDAT592),$ORI_TYPE = SORI_TYP(LCPDAT592),$APO = SAPO(LCPDAT592),$JERK = SJERK(LCPDAT592),$COLLMON_TOL_PRO[1] = USE_CM_PRO_VALUES(0)
;ENDFOLD

;FOLD SLIN P593 Vel=1 m/s CPDAT593 Tool[4]:Microflown3D Base[0];%{PE}
;FOLD Parameters ;%{h}
;Params IlfProvider=kukaroboter.basistech.inlineforms.movement.spline; Kuka.IsGlobalPoint=False; Kuka.PointName=P593; Kuka.BlendingEnabled=False; Kuka.MoveDataName=CPDAT593; Kuka.VelocityPath=1.000; Kuka.VelocityFieldEnabled=True; Kuka.ColDetectFieldEnabled=True; Kuka.CurrentCDSetIndex=0; Kuka.MovementParameterFieldEnabled=True; IlfCommand=SLIN
;ENDFOLD
SLIN XP593 WITH $VEL = SVEL_CP(2.0, , LCPDAT593),$TOOL = STOOL2(FP593),$BASE = SBASE(FP593.BASE_NO),$IPO_MODE = SIPO_MODE(FP593.IPO_FRAME),$LOAD = SLOAD(FP593.TOOL_NO),$ACC = SACC_CP(LCPDAT593),$ORI_TYPE = SORI_TYP(LCPDAT593),$APO = SAPO(LCPDAT593),$JERK = SJERK(LCPDAT593),$COLLMON_TOL_PRO[1] = USE_CM_PRO_VALUES(0)
;ENDFOLD

;FOLD SLIN P594 Vel=1 m/s CPDAT594 Tool[4]:Microflown3D Base[0];%{PE}
;FOLD Parameters ;%{h}
;Params IlfProvider=kukaroboter.basistech.inlineforms.movement.spline; Kuka.IsGlobalPoint=False; Kuka.PointName=P594; Kuka.BlendingEnabled=False; Kuka.MoveDataName=CPDAT594; Kuka.VelocityPath=1.000; Kuka.VelocityFieldEnabled=True; Kuka.ColDetectFieldEnabled=True; Kuka.CurrentCDSetIndex=0; Kuka.MovementParameterFieldEnabled=True; IlfCommand=SLIN
;ENDFOLD
SLIN XP594 WITH $VEL = SVEL_CP(2.0, , LCPDAT594),$TOOL = STOOL2(FP594),$BASE = SBASE(FP594.BASE_NO),$IPO_MODE = SIPO_MODE(FP594.IPO_FRAME),$LOAD = SLOAD(FP594.TOOL_NO),$ACC = SACC_CP(LCPDAT594),$ORI_TYPE = SORI_TYP(LCPDAT594),$APO = SAPO(LCPDAT594),$JERK = SJERK(LCPDAT594),$COLLMON_TOL_PRO[1] = USE_CM_PRO_VALUES(0)
;ENDFOLD

;FOLD SLIN P595 Vel=1 m/s CPDAT595 Tool[4]:Microflown3D Base[0];%{PE}
;FOLD Parameters ;%{h}
;Params IlfProvider=kukaroboter.basistech.inlineforms.movement.spline; Kuka.IsGlobalPoint=False; Kuka.PointName=P595; Kuka.BlendingEnabled=False; Kuka.MoveDataName=CPDAT595; Kuka.VelocityPath=1.000; Kuka.VelocityFieldEnabled=True; Kuka.ColDetectFieldEnabled=True; Kuka.CurrentCDSetIndex=0; Kuka.MovementParameterFieldEnabled=True; IlfCommand=SLIN
;ENDFOLD
SLIN XP595 WITH $VEL = SVEL_CP(2.0, , LCPDAT595),$TOOL = STOOL2(FP595),$BASE = SBASE(FP595.BASE_NO),$IPO_MODE = SIPO_MODE(FP595.IPO_FRAME),$LOAD = SLOAD(FP595.TOOL_NO),$ACC = SACC_CP(LCPDAT595),$ORI_TYPE = SORI_TYP(LCPDAT595),$APO = SAPO(LCPDAT595),$JERK = SJERK(LCPDAT595),$COLLMON_TOL_PRO[1] = USE_CM_PRO_VALUES(0)
;ENDFOLD

;FOLD SLIN P596 Vel=1 m/s CPDAT596 Tool[4]:Microflown3D Base[0];%{PE}
;FOLD Parameters ;%{h}
;Params IlfProvider=kukaroboter.basistech.inlineforms.movement.spline; Kuka.IsGlobalPoint=False; Kuka.PointName=P596; Kuka.BlendingEnabled=False; Kuka.MoveDataName=CPDAT596; Kuka.VelocityPath=1.000; Kuka.VelocityFieldEnabled=True; Kuka.ColDetectFieldEnabled=True; Kuka.CurrentCDSetIndex=0; Kuka.MovementParameterFieldEnabled=True; IlfCommand=SLIN
;ENDFOLD
SLIN XP596 WITH $VEL = SVEL_CP(2.0, , LCPDAT596),$TOOL = STOOL2(FP596),$BASE = SBASE(FP596.BASE_NO),$IPO_MODE = SIPO_MODE(FP596.IPO_FRAME),$LOAD = SLOAD(FP596.TOOL_NO),$ACC = SACC_CP(LCPDAT596),$ORI_TYPE = SORI_TYP(LCPDAT596),$APO = SAPO(LCPDAT596),$JERK = SJERK(LCPDAT596),$COLLMON_TOL_PRO[1] = USE_CM_PRO_VALUES(0)
;ENDFOLD

;FOLD SLIN P597 Vel=1 m/s CPDAT597 Tool[4]:Microflown3D Base[0];%{PE}
;FOLD Parameters ;%{h}
;Params IlfProvider=kukaroboter.basistech.inlineforms.movement.spline; Kuka.IsGlobalPoint=False; Kuka.PointName=P597; Kuka.BlendingEnabled=False; Kuka.MoveDataName=CPDAT597; Kuka.VelocityPath=1.000; Kuka.VelocityFieldEnabled=True; Kuka.ColDetectFieldEnabled=True; Kuka.CurrentCDSetIndex=0; Kuka.MovementParameterFieldEnabled=True; IlfCommand=SLIN
;ENDFOLD
SLIN XP597 WITH $VEL = SVEL_CP(2.0, , LCPDAT597),$TOOL = STOOL2(FP597),$BASE = SBASE(FP597.BASE_NO),$IPO_MODE = SIPO_MODE(FP597.IPO_FRAME),$LOAD = SLOAD(FP597.TOOL_NO),$ACC = SACC_CP(LCPDAT597),$ORI_TYPE = SORI_TYP(LCPDAT597),$APO = SAPO(LCPDAT597),$JERK = SJERK(LCPDAT597),$COLLMON_TOL_PRO[1] = USE_CM_PRO_VALUES(0)
;ENDFOLD

;FOLD SLIN P598 Vel=1 m/s CPDAT598 Tool[4]:Microflown3D Base[0];%{PE}
;FOLD Parameters ;%{h}
;Params IlfProvider=kukaroboter.basistech.inlineforms.movement.spline; Kuka.IsGlobalPoint=False; Kuka.PointName=P598; Kuka.BlendingEnabled=False; Kuka.MoveDataName=CPDAT598; Kuka.VelocityPath=1.000; Kuka.VelocityFieldEnabled=True; Kuka.ColDetectFieldEnabled=True; Kuka.CurrentCDSetIndex=0; Kuka.MovementParameterFieldEnabled=True; IlfCommand=SLIN
;ENDFOLD
SLIN XP598 WITH $VEL = SVEL_CP(2.0, , LCPDAT598),$TOOL = STOOL2(FP598),$BASE = SBASE(FP598.BASE_NO),$IPO_MODE = SIPO_MODE(FP598.IPO_FRAME),$LOAD = SLOAD(FP598.TOOL_NO),$ACC = SACC_CP(LCPDAT598),$ORI_TYPE = SORI_TYP(LCPDAT598),$APO = SAPO(LCPDAT598),$JERK = SJERK(LCPDAT598),$COLLMON_TOL_PRO[1] = USE_CM_PRO_VALUES(0)
;ENDFOLD

;FOLD SLIN P599 Vel=1 m/s CPDAT599 Tool[4]:Microflown3D Base[0];%{PE}
;FOLD Parameters ;%{h}
;Params IlfProvider=kukaroboter.basistech.inlineforms.movement.spline; Kuka.IsGlobalPoint=False; Kuka.PointName=P599; Kuka.BlendingEnabled=False; Kuka.MoveDataName=CPDAT599; Kuka.VelocityPath=1.000; Kuka.VelocityFieldEnabled=True; Kuka.ColDetectFieldEnabled=True; Kuka.CurrentCDSetIndex=0; Kuka.MovementParameterFieldEnabled=True; IlfCommand=SLIN
;ENDFOLD
SLIN XP599 WITH $VEL = SVEL_CP(2.0, , LCPDAT599),$TOOL = STOOL2(FP599),$BASE = SBASE(FP599.BASE_NO),$IPO_MODE = SIPO_MODE(FP599.IPO_FRAME),$LOAD = SLOAD(FP599.TOOL_NO),$ACC = SACC_CP(LCPDAT599),$ORI_TYPE = SORI_TYP(LCPDAT599),$APO = SAPO(LCPDAT599),$JERK = SJERK(LCPDAT599),$COLLMON_TOL_PRO[1] = USE_CM_PRO_VALUES(0)
;ENDFOLD

;FOLD SLIN P600 Vel=1 m/s CPDAT600 Tool[4]:Microflown3D Base[0];%{PE}
;FOLD Parameters ;%{h}
;Params IlfProvider=kukaroboter.basistech.inlineforms.movement.spline; Kuka.IsGlobalPoint=False; Kuka.PointName=P600; Kuka.BlendingEnabled=False; Kuka.MoveDataName=CPDAT600; Kuka.VelocityPath=1.000; Kuka.VelocityFieldEnabled=True; Kuka.ColDetectFieldEnabled=True; Kuka.CurrentCDSetIndex=0; Kuka.MovementParameterFieldEnabled=True; IlfCommand=SLIN
;ENDFOLD
SLIN XP600 WITH $VEL = SVEL_CP(2.0, , LCPDAT600),$TOOL = STOOL2(FP600),$BASE = SBASE(FP600.BASE_NO),$IPO_MODE = SIPO_MODE(FP600.IPO_FRAME),$LOAD = SLOAD(FP600.TOOL_NO),$ACC = SACC_CP(LCPDAT600),$ORI_TYPE = SORI_TYP(LCPDAT600),$APO = SAPO(LCPDAT600),$JERK = SJERK(LCPDAT600),$COLLMON_TOL_PRO[1] = USE_CM_PRO_VALUES(0)
;ENDFOLD

;FOLD SLIN P601 Vel=1 m/s CPDAT601 Tool[4]:Microflown3D Base[0];%{PE}
;FOLD Parameters ;%{h}
;Params IlfProvider=kukaroboter.basistech.inlineforms.movement.spline; Kuka.IsGlobalPoint=False; Kuka.PointName=P601; Kuka.BlendingEnabled=False; Kuka.MoveDataName=CPDAT601; Kuka.VelocityPath=1.000; Kuka.VelocityFieldEnabled=True; Kuka.ColDetectFieldEnabled=True; Kuka.CurrentCDSetIndex=0; Kuka.MovementParameterFieldEnabled=True; IlfCommand=SLIN
;ENDFOLD
SLIN XP601 WITH $VEL = SVEL_CP(2.0, , LCPDAT601),$TOOL = STOOL2(FP601),$BASE = SBASE(FP601.BASE_NO),$IPO_MODE = SIPO_MODE(FP601.IPO_FRAME),$LOAD = SLOAD(FP601.TOOL_NO),$ACC = SACC_CP(LCPDAT601),$ORI_TYPE = SORI_TYP(LCPDAT601),$APO = SAPO(LCPDAT601),$JERK = SJERK(LCPDAT601),$COLLMON_TOL_PRO[1] = USE_CM_PRO_VALUES(0)
;ENDFOLD

;FOLD SLIN P602 Vel=1 m/s CPDAT602 Tool[4]:Microflown3D Base[0];%{PE}
;FOLD Parameters ;%{h}
;Params IlfProvider=kukaroboter.basistech.inlineforms.movement.spline; Kuka.IsGlobalPoint=False; Kuka.PointName=P602; Kuka.BlendingEnabled=False; Kuka.MoveDataName=CPDAT602; Kuka.VelocityPath=1.000; Kuka.VelocityFieldEnabled=True; Kuka.ColDetectFieldEnabled=True; Kuka.CurrentCDSetIndex=0; Kuka.MovementParameterFieldEnabled=True; IlfCommand=SLIN
;ENDFOLD
SLIN XP602 WITH $VEL = SVEL_CP(2.0, , LCPDAT602),$TOOL = STOOL2(FP602),$BASE = SBASE(FP602.BASE_NO),$IPO_MODE = SIPO_MODE(FP602.IPO_FRAME),$LOAD = SLOAD(FP602.TOOL_NO),$ACC = SACC_CP(LCPDAT602),$ORI_TYPE = SORI_TYP(LCPDAT602),$APO = SAPO(LCPDAT602),$JERK = SJERK(LCPDAT602),$COLLMON_TOL_PRO[1] = USE_CM_PRO_VALUES(0)
;ENDFOLD

;FOLD SLIN P603 Vel=1 m/s CPDAT603 Tool[4]:Microflown3D Base[0];%{PE}
;FOLD Parameters ;%{h}
;Params IlfProvider=kukaroboter.basistech.inlineforms.movement.spline; Kuka.IsGlobalPoint=False; Kuka.PointName=P603; Kuka.BlendingEnabled=False; Kuka.MoveDataName=CPDAT603; Kuka.VelocityPath=1.000; Kuka.VelocityFieldEnabled=True; Kuka.ColDetectFieldEnabled=True; Kuka.CurrentCDSetIndex=0; Kuka.MovementParameterFieldEnabled=True; IlfCommand=SLIN
;ENDFOLD
SLIN XP603 WITH $VEL = SVEL_CP(2.0, , LCPDAT603),$TOOL = STOOL2(FP603),$BASE = SBASE(FP603.BASE_NO),$IPO_MODE = SIPO_MODE(FP603.IPO_FRAME),$LOAD = SLOAD(FP603.TOOL_NO),$ACC = SACC_CP(LCPDAT603),$ORI_TYPE = SORI_TYP(LCPDAT603),$APO = SAPO(LCPDAT603),$JERK = SJERK(LCPDAT603),$COLLMON_TOL_PRO[1] = USE_CM_PRO_VALUES(0)
;ENDFOLD

;FOLD SLIN P604 Vel=1 m/s CPDAT604 Tool[4]:Microflown3D Base[0];%{PE}
;FOLD Parameters ;%{h}
;Params IlfProvider=kukaroboter.basistech.inlineforms.movement.spline; Kuka.IsGlobalPoint=False; Kuka.PointName=P604; Kuka.BlendingEnabled=False; Kuka.MoveDataName=CPDAT604; Kuka.VelocityPath=1.000; Kuka.VelocityFieldEnabled=True; Kuka.ColDetectFieldEnabled=True; Kuka.CurrentCDSetIndex=0; Kuka.MovementParameterFieldEnabled=True; IlfCommand=SLIN
;ENDFOLD
SLIN XP604 WITH $VEL = SVEL_CP(2.0, , LCPDAT604),$TOOL = STOOL2(FP604),$BASE = SBASE(FP604.BASE_NO),$IPO_MODE = SIPO_MODE(FP604.IPO_FRAME),$LOAD = SLOAD(FP604.TOOL_NO),$ACC = SACC_CP(LCPDAT604),$ORI_TYPE = SORI_TYP(LCPDAT604),$APO = SAPO(LCPDAT604),$JERK = SJERK(LCPDAT604),$COLLMON_TOL_PRO[1] = USE_CM_PRO_VALUES(0)
;ENDFOLD

;FOLD SLIN P605 Vel=1 m/s CPDAT605 Tool[4]:Microflown3D Base[0];%{PE}
;FOLD Parameters ;%{h}
;Params IlfProvider=kukaroboter.basistech.inlineforms.movement.spline; Kuka.IsGlobalPoint=False; Kuka.PointName=P605; Kuka.BlendingEnabled=False; Kuka.MoveDataName=CPDAT605; Kuka.VelocityPath=1.000; Kuka.VelocityFieldEnabled=True; Kuka.ColDetectFieldEnabled=True; Kuka.CurrentCDSetIndex=0; Kuka.MovementParameterFieldEnabled=True; IlfCommand=SLIN
;ENDFOLD
SLIN XP605 WITH $VEL = SVEL_CP(2.0, , LCPDAT605),$TOOL = STOOL2(FP605),$BASE = SBASE(FP605.BASE_NO),$IPO_MODE = SIPO_MODE(FP605.IPO_FRAME),$LOAD = SLOAD(FP605.TOOL_NO),$ACC = SACC_CP(LCPDAT605),$ORI_TYPE = SORI_TYP(LCPDAT605),$APO = SAPO(LCPDAT605),$JERK = SJERK(LCPDAT605),$COLLMON_TOL_PRO[1] = USE_CM_PRO_VALUES(0)
;ENDFOLD

;FOLD SLIN P606 Vel=1 m/s CPDAT606 Tool[4]:Microflown3D Base[0];%{PE}
;FOLD Parameters ;%{h}
;Params IlfProvider=kukaroboter.basistech.inlineforms.movement.spline; Kuka.IsGlobalPoint=False; Kuka.PointName=P606; Kuka.BlendingEnabled=False; Kuka.MoveDataName=CPDAT606; Kuka.VelocityPath=1.000; Kuka.VelocityFieldEnabled=True; Kuka.ColDetectFieldEnabled=True; Kuka.CurrentCDSetIndex=0; Kuka.MovementParameterFieldEnabled=True; IlfCommand=SLIN
;ENDFOLD
SLIN XP606 WITH $VEL = SVEL_CP(2.0, , LCPDAT606),$TOOL = STOOL2(FP606),$BASE = SBASE(FP606.BASE_NO),$IPO_MODE = SIPO_MODE(FP606.IPO_FRAME),$LOAD = SLOAD(FP606.TOOL_NO),$ACC = SACC_CP(LCPDAT606),$ORI_TYPE = SORI_TYP(LCPDAT606),$APO = SAPO(LCPDAT606),$JERK = SJERK(LCPDAT606),$COLLMON_TOL_PRO[1] = USE_CM_PRO_VALUES(0)
;ENDFOLD

;FOLD SLIN P607 Vel=1 m/s CPDAT607 Tool[4]:Microflown3D Base[0];%{PE}
;FOLD Parameters ;%{h}
;Params IlfProvider=kukaroboter.basistech.inlineforms.movement.spline; Kuka.IsGlobalPoint=False; Kuka.PointName=P607; Kuka.BlendingEnabled=False; Kuka.MoveDataName=CPDAT607; Kuka.VelocityPath=1.000; Kuka.VelocityFieldEnabled=True; Kuka.ColDetectFieldEnabled=True; Kuka.CurrentCDSetIndex=0; Kuka.MovementParameterFieldEnabled=True; IlfCommand=SLIN
;ENDFOLD
SLIN XP607 WITH $VEL = SVEL_CP(2.0, , LCPDAT607),$TOOL = STOOL2(FP607),$BASE = SBASE(FP607.BASE_NO),$IPO_MODE = SIPO_MODE(FP607.IPO_FRAME),$LOAD = SLOAD(FP607.TOOL_NO),$ACC = SACC_CP(LCPDAT607),$ORI_TYPE = SORI_TYP(LCPDAT607),$APO = SAPO(LCPDAT607),$JERK = SJERK(LCPDAT607),$COLLMON_TOL_PRO[1] = USE_CM_PRO_VALUES(0)
;ENDFOLD

;FOLD SLIN P608 Vel=1 m/s CPDAT608 Tool[4]:Microflown3D Base[0];%{PE}
;FOLD Parameters ;%{h}
;Params IlfProvider=kukaroboter.basistech.inlineforms.movement.spline; Kuka.IsGlobalPoint=False; Kuka.PointName=P608; Kuka.BlendingEnabled=False; Kuka.MoveDataName=CPDAT608; Kuka.VelocityPath=1.000; Kuka.VelocityFieldEnabled=True; Kuka.ColDetectFieldEnabled=True; Kuka.CurrentCDSetIndex=0; Kuka.MovementParameterFieldEnabled=True; IlfCommand=SLIN
;ENDFOLD
SLIN XP608 WITH $VEL = SVEL_CP(2.0, , LCPDAT608),$TOOL = STOOL2(FP608),$BASE = SBASE(FP608.BASE_NO),$IPO_MODE = SIPO_MODE(FP608.IPO_FRAME),$LOAD = SLOAD(FP608.TOOL_NO),$ACC = SACC_CP(LCPDAT608),$ORI_TYPE = SORI_TYP(LCPDAT608),$APO = SAPO(LCPDAT608),$JERK = SJERK(LCPDAT608),$COLLMON_TOL_PRO[1] = USE_CM_PRO_VALUES(0)
;ENDFOLD

;FOLD SLIN P609 Vel=1 m/s CPDAT609 Tool[4]:Microflown3D Base[0];%{PE}
;FOLD Parameters ;%{h}
;Params IlfProvider=kukaroboter.basistech.inlineforms.movement.spline; Kuka.IsGlobalPoint=False; Kuka.PointName=P609; Kuka.BlendingEnabled=False; Kuka.MoveDataName=CPDAT609; Kuka.VelocityPath=1.000; Kuka.VelocityFieldEnabled=True; Kuka.ColDetectFieldEnabled=True; Kuka.CurrentCDSetIndex=0; Kuka.MovementParameterFieldEnabled=True; IlfCommand=SLIN
;ENDFOLD
SLIN XP609 WITH $VEL = SVEL_CP(2.0, , LCPDAT609),$TOOL = STOOL2(FP609),$BASE = SBASE(FP609.BASE_NO),$IPO_MODE = SIPO_MODE(FP609.IPO_FRAME),$LOAD = SLOAD(FP609.TOOL_NO),$ACC = SACC_CP(LCPDAT609),$ORI_TYPE = SORI_TYP(LCPDAT609),$APO = SAPO(LCPDAT609),$JERK = SJERK(LCPDAT609),$COLLMON_TOL_PRO[1] = USE_CM_PRO_VALUES(0)
;ENDFOLD

;FOLD SLIN P610 Vel=1 m/s CPDAT610 Tool[4]:Microflown3D Base[0];%{PE}
;FOLD Parameters ;%{h}
;Params IlfProvider=kukaroboter.basistech.inlineforms.movement.spline; Kuka.IsGlobalPoint=False; Kuka.PointName=P610; Kuka.BlendingEnabled=False; Kuka.MoveDataName=CPDAT610; Kuka.VelocityPath=1.000; Kuka.VelocityFieldEnabled=True; Kuka.ColDetectFieldEnabled=True; Kuka.CurrentCDSetIndex=0; Kuka.MovementParameterFieldEnabled=True; IlfCommand=SLIN
;ENDFOLD
SLIN XP610 WITH $VEL = SVEL_CP(2.0, , LCPDAT610),$TOOL = STOOL2(FP610),$BASE = SBASE(FP610.BASE_NO),$IPO_MODE = SIPO_MODE(FP610.IPO_FRAME),$LOAD = SLOAD(FP610.TOOL_NO),$ACC = SACC_CP(LCPDAT610),$ORI_TYPE = SORI_TYP(LCPDAT610),$APO = SAPO(LCPDAT610),$JERK = SJERK(LCPDAT610),$COLLMON_TOL_PRO[1] = USE_CM_PRO_VALUES(0)
;ENDFOLD

;FOLD SLIN P611 Vel=1 m/s CPDAT611 Tool[4]:Microflown3D Base[0];%{PE}
;FOLD Parameters ;%{h}
;Params IlfProvider=kukaroboter.basistech.inlineforms.movement.spline; Kuka.IsGlobalPoint=False; Kuka.PointName=P611; Kuka.BlendingEnabled=False; Kuka.MoveDataName=CPDAT611; Kuka.VelocityPath=1.000; Kuka.VelocityFieldEnabled=True; Kuka.ColDetectFieldEnabled=True; Kuka.CurrentCDSetIndex=0; Kuka.MovementParameterFieldEnabled=True; IlfCommand=SLIN
;ENDFOLD
SLIN XP611 WITH $VEL = SVEL_CP(2.0, , LCPDAT611),$TOOL = STOOL2(FP611),$BASE = SBASE(FP611.BASE_NO),$IPO_MODE = SIPO_MODE(FP611.IPO_FRAME),$LOAD = SLOAD(FP611.TOOL_NO),$ACC = SACC_CP(LCPDAT611),$ORI_TYPE = SORI_TYP(LCPDAT611),$APO = SAPO(LCPDAT611),$JERK = SJERK(LCPDAT611),$COLLMON_TOL_PRO[1] = USE_CM_PRO_VALUES(0)
;ENDFOLD

;FOLD SLIN P612 Vel=1 m/s CPDAT612 Tool[4]:Microflown3D Base[0];%{PE}
;FOLD Parameters ;%{h}
;Params IlfProvider=kukaroboter.basistech.inlineforms.movement.spline; Kuka.IsGlobalPoint=False; Kuka.PointName=P612; Kuka.BlendingEnabled=False; Kuka.MoveDataName=CPDAT612; Kuka.VelocityPath=1.000; Kuka.VelocityFieldEnabled=True; Kuka.ColDetectFieldEnabled=True; Kuka.CurrentCDSetIndex=0; Kuka.MovementParameterFieldEnabled=True; IlfCommand=SLIN
;ENDFOLD
SLIN XP612 WITH $VEL = SVEL_CP(2.0, , LCPDAT612),$TOOL = STOOL2(FP612),$BASE = SBASE(FP612.BASE_NO),$IPO_MODE = SIPO_MODE(FP612.IPO_FRAME),$LOAD = SLOAD(FP612.TOOL_NO),$ACC = SACC_CP(LCPDAT612),$ORI_TYPE = SORI_TYP(LCPDAT612),$APO = SAPO(LCPDAT612),$JERK = SJERK(LCPDAT612),$COLLMON_TOL_PRO[1] = USE_CM_PRO_VALUES(0)
;ENDFOLD

;FOLD SLIN P613 Vel=1 m/s CPDAT613 Tool[4]:Microflown3D Base[0];%{PE}
;FOLD Parameters ;%{h}
;Params IlfProvider=kukaroboter.basistech.inlineforms.movement.spline; Kuka.IsGlobalPoint=False; Kuka.PointName=P613; Kuka.BlendingEnabled=False; Kuka.MoveDataName=CPDAT613; Kuka.VelocityPath=1.000; Kuka.VelocityFieldEnabled=True; Kuka.ColDetectFieldEnabled=True; Kuka.CurrentCDSetIndex=0; Kuka.MovementParameterFieldEnabled=True; IlfCommand=SLIN
;ENDFOLD
SLIN XP613 WITH $VEL = SVEL_CP(2.0, , LCPDAT613),$TOOL = STOOL2(FP613),$BASE = SBASE(FP613.BASE_NO),$IPO_MODE = SIPO_MODE(FP613.IPO_FRAME),$LOAD = SLOAD(FP613.TOOL_NO),$ACC = SACC_CP(LCPDAT613),$ORI_TYPE = SORI_TYP(LCPDAT613),$APO = SAPO(LCPDAT613),$JERK = SJERK(LCPDAT613),$COLLMON_TOL_PRO[1] = USE_CM_PRO_VALUES(0)
;ENDFOLD

;FOLD SLIN P614 Vel=1 m/s CPDAT614 Tool[4]:Microflown3D Base[0];%{PE}
;FOLD Parameters ;%{h}
;Params IlfProvider=kukaroboter.basistech.inlineforms.movement.spline; Kuka.IsGlobalPoint=False; Kuka.PointName=P614; Kuka.BlendingEnabled=False; Kuka.MoveDataName=CPDAT614; Kuka.VelocityPath=1.000; Kuka.VelocityFieldEnabled=True; Kuka.ColDetectFieldEnabled=True; Kuka.CurrentCDSetIndex=0; Kuka.MovementParameterFieldEnabled=True; IlfCommand=SLIN
;ENDFOLD
SLIN XP614 WITH $VEL = SVEL_CP(2.0, , LCPDAT614),$TOOL = STOOL2(FP614),$BASE = SBASE(FP614.BASE_NO),$IPO_MODE = SIPO_MODE(FP614.IPO_FRAME),$LOAD = SLOAD(FP614.TOOL_NO),$ACC = SACC_CP(LCPDAT614),$ORI_TYPE = SORI_TYP(LCPDAT614),$APO = SAPO(LCPDAT614),$JERK = SJERK(LCPDAT614),$COLLMON_TOL_PRO[1] = USE_CM_PRO_VALUES(0)
;ENDFOLD

;FOLD SLIN P615 Vel=1 m/s CPDAT615 Tool[4]:Microflown3D Base[0];%{PE}
;FOLD Parameters ;%{h}
;Params IlfProvider=kukaroboter.basistech.inlineforms.movement.spline; Kuka.IsGlobalPoint=False; Kuka.PointName=P615; Kuka.BlendingEnabled=False; Kuka.MoveDataName=CPDAT615; Kuka.VelocityPath=1.000; Kuka.VelocityFieldEnabled=True; Kuka.ColDetectFieldEnabled=True; Kuka.CurrentCDSetIndex=0; Kuka.MovementParameterFieldEnabled=True; IlfCommand=SLIN
;ENDFOLD
SLIN XP615 WITH $VEL = SVEL_CP(2.0, , LCPDAT615),$TOOL = STOOL2(FP615),$BASE = SBASE(FP615.BASE_NO),$IPO_MODE = SIPO_MODE(FP615.IPO_FRAME),$LOAD = SLOAD(FP615.TOOL_NO),$ACC = SACC_CP(LCPDAT615),$ORI_TYPE = SORI_TYP(LCPDAT615),$APO = SAPO(LCPDAT615),$JERK = SJERK(LCPDAT615),$COLLMON_TOL_PRO[1] = USE_CM_PRO_VALUES(0)
;ENDFOLD

;FOLD SLIN P616 Vel=1 m/s CPDAT616 Tool[4]:Microflown3D Base[0];%{PE}
;FOLD Parameters ;%{h}
;Params IlfProvider=kukaroboter.basistech.inlineforms.movement.spline; Kuka.IsGlobalPoint=False; Kuka.PointName=P616; Kuka.BlendingEnabled=False; Kuka.MoveDataName=CPDAT616; Kuka.VelocityPath=1.000; Kuka.VelocityFieldEnabled=True; Kuka.ColDetectFieldEnabled=True; Kuka.CurrentCDSetIndex=0; Kuka.MovementParameterFieldEnabled=True; IlfCommand=SLIN
;ENDFOLD
SLIN XP616 WITH $VEL = SVEL_CP(2.0, , LCPDAT616),$TOOL = STOOL2(FP616),$BASE = SBASE(FP616.BASE_NO),$IPO_MODE = SIPO_MODE(FP616.IPO_FRAME),$LOAD = SLOAD(FP616.TOOL_NO),$ACC = SACC_CP(LCPDAT616),$ORI_TYPE = SORI_TYP(LCPDAT616),$APO = SAPO(LCPDAT616),$JERK = SJERK(LCPDAT616),$COLLMON_TOL_PRO[1] = USE_CM_PRO_VALUES(0)
;ENDFOLD

;FOLD SLIN P617 Vel=1 m/s CPDAT617 Tool[4]:Microflown3D Base[0];%{PE}
;FOLD Parameters ;%{h}
;Params IlfProvider=kukaroboter.basistech.inlineforms.movement.spline; Kuka.IsGlobalPoint=False; Kuka.PointName=P617; Kuka.BlendingEnabled=False; Kuka.MoveDataName=CPDAT617; Kuka.VelocityPath=1.000; Kuka.VelocityFieldEnabled=True; Kuka.ColDetectFieldEnabled=True; Kuka.CurrentCDSetIndex=0; Kuka.MovementParameterFieldEnabled=True; IlfCommand=SLIN
;ENDFOLD
SLIN XP617 WITH $VEL = SVEL_CP(2.0, , LCPDAT617),$TOOL = STOOL2(FP617),$BASE = SBASE(FP617.BASE_NO),$IPO_MODE = SIPO_MODE(FP617.IPO_FRAME),$LOAD = SLOAD(FP617.TOOL_NO),$ACC = SACC_CP(LCPDAT617),$ORI_TYPE = SORI_TYP(LCPDAT617),$APO = SAPO(LCPDAT617),$JERK = SJERK(LCPDAT617),$COLLMON_TOL_PRO[1] = USE_CM_PRO_VALUES(0)
;ENDFOLD

;FOLD SLIN P618 Vel=1 m/s CPDAT618 Tool[4]:Microflown3D Base[0];%{PE}
;FOLD Parameters ;%{h}
;Params IlfProvider=kukaroboter.basistech.inlineforms.movement.spline; Kuka.IsGlobalPoint=False; Kuka.PointName=P618; Kuka.BlendingEnabled=False; Kuka.MoveDataName=CPDAT618; Kuka.VelocityPath=1.000; Kuka.VelocityFieldEnabled=True; Kuka.ColDetectFieldEnabled=True; Kuka.CurrentCDSetIndex=0; Kuka.MovementParameterFieldEnabled=True; IlfCommand=SLIN
;ENDFOLD
SLIN XP618 WITH $VEL = SVEL_CP(2.0, , LCPDAT618),$TOOL = STOOL2(FP618),$BASE = SBASE(FP618.BASE_NO),$IPO_MODE = SIPO_MODE(FP618.IPO_FRAME),$LOAD = SLOAD(FP618.TOOL_NO),$ACC = SACC_CP(LCPDAT618),$ORI_TYPE = SORI_TYP(LCPDAT618),$APO = SAPO(LCPDAT618),$JERK = SJERK(LCPDAT618),$COLLMON_TOL_PRO[1] = USE_CM_PRO_VALUES(0)
;ENDFOLD

;FOLD SLIN P619 Vel=1 m/s CPDAT619 Tool[4]:Microflown3D Base[0];%{PE}
;FOLD Parameters ;%{h}
;Params IlfProvider=kukaroboter.basistech.inlineforms.movement.spline; Kuka.IsGlobalPoint=False; Kuka.PointName=P619; Kuka.BlendingEnabled=False; Kuka.MoveDataName=CPDAT619; Kuka.VelocityPath=1.000; Kuka.VelocityFieldEnabled=True; Kuka.ColDetectFieldEnabled=True; Kuka.CurrentCDSetIndex=0; Kuka.MovementParameterFieldEnabled=True; IlfCommand=SLIN
;ENDFOLD
SLIN XP619 WITH $VEL = SVEL_CP(2.0, , LCPDAT619),$TOOL = STOOL2(FP619),$BASE = SBASE(FP619.BASE_NO),$IPO_MODE = SIPO_MODE(FP619.IPO_FRAME),$LOAD = SLOAD(FP619.TOOL_NO),$ACC = SACC_CP(LCPDAT619),$ORI_TYPE = SORI_TYP(LCPDAT619),$APO = SAPO(LCPDAT619),$JERK = SJERK(LCPDAT619),$COLLMON_TOL_PRO[1] = USE_CM_PRO_VALUES(0)
;ENDFOLD

;FOLD SLIN P620 Vel=1 m/s CPDAT620 Tool[4]:Microflown3D Base[0];%{PE}
;FOLD Parameters ;%{h}
;Params IlfProvider=kukaroboter.basistech.inlineforms.movement.spline; Kuka.IsGlobalPoint=False; Kuka.PointName=P620; Kuka.BlendingEnabled=False; Kuka.MoveDataName=CPDAT620; Kuka.VelocityPath=1.000; Kuka.VelocityFieldEnabled=True; Kuka.ColDetectFieldEnabled=True; Kuka.CurrentCDSetIndex=0; Kuka.MovementParameterFieldEnabled=True; IlfCommand=SLIN
;ENDFOLD
SLIN XP620 WITH $VEL = SVEL_CP(2.0, , LCPDAT620),$TOOL = STOOL2(FP620),$BASE = SBASE(FP620.BASE_NO),$IPO_MODE = SIPO_MODE(FP620.IPO_FRAME),$LOAD = SLOAD(FP620.TOOL_NO),$ACC = SACC_CP(LCPDAT620),$ORI_TYPE = SORI_TYP(LCPDAT620),$APO = SAPO(LCPDAT620),$JERK = SJERK(LCPDAT620),$COLLMON_TOL_PRO[1] = USE_CM_PRO_VALUES(0)
;ENDFOLD

;FOLD SLIN P621 Vel=1 m/s CPDAT621 Tool[4]:Microflown3D Base[0];%{PE}
;FOLD Parameters ;%{h}
;Params IlfProvider=kukaroboter.basistech.inlineforms.movement.spline; Kuka.IsGlobalPoint=False; Kuka.PointName=P621; Kuka.BlendingEnabled=False; Kuka.MoveDataName=CPDAT621; Kuka.VelocityPath=1.000; Kuka.VelocityFieldEnabled=True; Kuka.ColDetectFieldEnabled=True; Kuka.CurrentCDSetIndex=0; Kuka.MovementParameterFieldEnabled=True; IlfCommand=SLIN
;ENDFOLD
SLIN XP621 WITH $VEL = SVEL_CP(2.0, , LCPDAT621),$TOOL = STOOL2(FP621),$BASE = SBASE(FP621.BASE_NO),$IPO_MODE = SIPO_MODE(FP621.IPO_FRAME),$LOAD = SLOAD(FP621.TOOL_NO),$ACC = SACC_CP(LCPDAT621),$ORI_TYPE = SORI_TYP(LCPDAT621),$APO = SAPO(LCPDAT621),$JERK = SJERK(LCPDAT621),$COLLMON_TOL_PRO[1] = USE_CM_PRO_VALUES(0)
;ENDFOLD

;FOLD SLIN P622 Vel=1 m/s CPDAT622 Tool[4]:Microflown3D Base[0];%{PE}
;FOLD Parameters ;%{h}
;Params IlfProvider=kukaroboter.basistech.inlineforms.movement.spline; Kuka.IsGlobalPoint=False; Kuka.PointName=P622; Kuka.BlendingEnabled=False; Kuka.MoveDataName=CPDAT622; Kuka.VelocityPath=1.000; Kuka.VelocityFieldEnabled=True; Kuka.ColDetectFieldEnabled=True; Kuka.CurrentCDSetIndex=0; Kuka.MovementParameterFieldEnabled=True; IlfCommand=SLIN
;ENDFOLD
SLIN XP622 WITH $VEL = SVEL_CP(2.0, , LCPDAT622),$TOOL = STOOL2(FP622),$BASE = SBASE(FP622.BASE_NO),$IPO_MODE = SIPO_MODE(FP622.IPO_FRAME),$LOAD = SLOAD(FP622.TOOL_NO),$ACC = SACC_CP(LCPDAT622),$ORI_TYPE = SORI_TYP(LCPDAT622),$APO = SAPO(LCPDAT622),$JERK = SJERK(LCPDAT622),$COLLMON_TOL_PRO[1] = USE_CM_PRO_VALUES(0)
;ENDFOLD

;FOLD SLIN P623 Vel=1 m/s CPDAT623 Tool[4]:Microflown3D Base[0];%{PE}
;FOLD Parameters ;%{h}
;Params IlfProvider=kukaroboter.basistech.inlineforms.movement.spline; Kuka.IsGlobalPoint=False; Kuka.PointName=P623; Kuka.BlendingEnabled=False; Kuka.MoveDataName=CPDAT623; Kuka.VelocityPath=1.000; Kuka.VelocityFieldEnabled=True; Kuka.ColDetectFieldEnabled=True; Kuka.CurrentCDSetIndex=0; Kuka.MovementParameterFieldEnabled=True; IlfCommand=SLIN
;ENDFOLD
SLIN XP623 WITH $VEL = SVEL_CP(2.0, , LCPDAT623),$TOOL = STOOL2(FP623),$BASE = SBASE(FP623.BASE_NO),$IPO_MODE = SIPO_MODE(FP623.IPO_FRAME),$LOAD = SLOAD(FP623.TOOL_NO),$ACC = SACC_CP(LCPDAT623),$ORI_TYPE = SORI_TYP(LCPDAT623),$APO = SAPO(LCPDAT623),$JERK = SJERK(LCPDAT623),$COLLMON_TOL_PRO[1] = USE_CM_PRO_VALUES(0)
;ENDFOLD

;FOLD SLIN P624 Vel=1 m/s CPDAT624 Tool[4]:Microflown3D Base[0];%{PE}
;FOLD Parameters ;%{h}
;Params IlfProvider=kukaroboter.basistech.inlineforms.movement.spline; Kuka.IsGlobalPoint=False; Kuka.PointName=P624; Kuka.BlendingEnabled=False; Kuka.MoveDataName=CPDAT624; Kuka.VelocityPath=1.000; Kuka.VelocityFieldEnabled=True; Kuka.ColDetectFieldEnabled=True; Kuka.CurrentCDSetIndex=0; Kuka.MovementParameterFieldEnabled=True; IlfCommand=SLIN
;ENDFOLD
SLIN XP624 WITH $VEL = SVEL_CP(2.0, , LCPDAT624),$TOOL = STOOL2(FP624),$BASE = SBASE(FP624.BASE_NO),$IPO_MODE = SIPO_MODE(FP624.IPO_FRAME),$LOAD = SLOAD(FP624.TOOL_NO),$ACC = SACC_CP(LCPDAT624),$ORI_TYPE = SORI_TYP(LCPDAT624),$APO = SAPO(LCPDAT624),$JERK = SJERK(LCPDAT624),$COLLMON_TOL_PRO[1] = USE_CM_PRO_VALUES(0)
;ENDFOLD

;FOLD SLIN P625 Vel=1 m/s CPDAT625 Tool[4]:Microflown3D Base[0];%{PE}
;FOLD Parameters ;%{h}
;Params IlfProvider=kukaroboter.basistech.inlineforms.movement.spline; Kuka.IsGlobalPoint=False; Kuka.PointName=P625; Kuka.BlendingEnabled=False; Kuka.MoveDataName=CPDAT625; Kuka.VelocityPath=1.000; Kuka.VelocityFieldEnabled=True; Kuka.ColDetectFieldEnabled=True; Kuka.CurrentCDSetIndex=0; Kuka.MovementParameterFieldEnabled=True; IlfCommand=SLIN
;ENDFOLD
SLIN XP625 WITH $VEL = SVEL_CP(2.0, , LCPDAT625),$TOOL = STOOL2(FP625),$BASE = SBASE(FP625.BASE_NO),$IPO_MODE = SIPO_MODE(FP625.IPO_FRAME),$LOAD = SLOAD(FP625.TOOL_NO),$ACC = SACC_CP(LCPDAT625),$ORI_TYPE = SORI_TYP(LCPDAT625),$APO = SAPO(LCPDAT625),$JERK = SJERK(LCPDAT625),$COLLMON_TOL_PRO[1] = USE_CM_PRO_VALUES(0)
;ENDFOLD

;FOLD SLIN P626 Vel=1 m/s CPDAT626 Tool[4]:Microflown3D Base[0];%{PE}
;FOLD Parameters ;%{h}
;Params IlfProvider=kukaroboter.basistech.inlineforms.movement.spline; Kuka.IsGlobalPoint=False; Kuka.PointName=P626; Kuka.BlendingEnabled=False; Kuka.MoveDataName=CPDAT626; Kuka.VelocityPath=1.000; Kuka.VelocityFieldEnabled=True; Kuka.ColDetectFieldEnabled=True; Kuka.CurrentCDSetIndex=0; Kuka.MovementParameterFieldEnabled=True; IlfCommand=SLIN
;ENDFOLD
SLIN XP626 WITH $VEL = SVEL_CP(2.0, , LCPDAT626),$TOOL = STOOL2(FP626),$BASE = SBASE(FP626.BASE_NO),$IPO_MODE = SIPO_MODE(FP626.IPO_FRAME),$LOAD = SLOAD(FP626.TOOL_NO),$ACC = SACC_CP(LCPDAT626),$ORI_TYPE = SORI_TYP(LCPDAT626),$APO = SAPO(LCPDAT626),$JERK = SJERK(LCPDAT626),$COLLMON_TOL_PRO[1] = USE_CM_PRO_VALUES(0)
;ENDFOLD

;FOLD SLIN P627 Vel=1 m/s CPDAT627 Tool[4]:Microflown3D Base[0];%{PE}
;FOLD Parameters ;%{h}
;Params IlfProvider=kukaroboter.basistech.inlineforms.movement.spline; Kuka.IsGlobalPoint=False; Kuka.PointName=P627; Kuka.BlendingEnabled=False; Kuka.MoveDataName=CPDAT627; Kuka.VelocityPath=1.000; Kuka.VelocityFieldEnabled=True; Kuka.ColDetectFieldEnabled=True; Kuka.CurrentCDSetIndex=0; Kuka.MovementParameterFieldEnabled=True; IlfCommand=SLIN
;ENDFOLD
SLIN XP627 WITH $VEL = SVEL_CP(2.0, , LCPDAT627),$TOOL = STOOL2(FP627),$BASE = SBASE(FP627.BASE_NO),$IPO_MODE = SIPO_MODE(FP627.IPO_FRAME),$LOAD = SLOAD(FP627.TOOL_NO),$ACC = SACC_CP(LCPDAT627),$ORI_TYPE = SORI_TYP(LCPDAT627),$APO = SAPO(LCPDAT627),$JERK = SJERK(LCPDAT627),$COLLMON_TOL_PRO[1] = USE_CM_PRO_VALUES(0)
;ENDFOLD

;FOLD SLIN P628 Vel=1 m/s CPDAT628 Tool[4]:Microflown3D Base[0];%{PE}
;FOLD Parameters ;%{h}
;Params IlfProvider=kukaroboter.basistech.inlineforms.movement.spline; Kuka.IsGlobalPoint=False; Kuka.PointName=P628; Kuka.BlendingEnabled=False; Kuka.MoveDataName=CPDAT628; Kuka.VelocityPath=1.000; Kuka.VelocityFieldEnabled=True; Kuka.ColDetectFieldEnabled=True; Kuka.CurrentCDSetIndex=0; Kuka.MovementParameterFieldEnabled=True; IlfCommand=SLIN
;ENDFOLD
SLIN XP628 WITH $VEL = SVEL_CP(2.0, , LCPDAT628),$TOOL = STOOL2(FP628),$BASE = SBASE(FP628.BASE_NO),$IPO_MODE = SIPO_MODE(FP628.IPO_FRAME),$LOAD = SLOAD(FP628.TOOL_NO),$ACC = SACC_CP(LCPDAT628),$ORI_TYPE = SORI_TYP(LCPDAT628),$APO = SAPO(LCPDAT628),$JERK = SJERK(LCPDAT628),$COLLMON_TOL_PRO[1] = USE_CM_PRO_VALUES(0)
;ENDFOLD

;FOLD SLIN P629 Vel=1 m/s CPDAT629 Tool[4]:Microflown3D Base[0];%{PE}
;FOLD Parameters ;%{h}
;Params IlfProvider=kukaroboter.basistech.inlineforms.movement.spline; Kuka.IsGlobalPoint=False; Kuka.PointName=P629; Kuka.BlendingEnabled=False; Kuka.MoveDataName=CPDAT629; Kuka.VelocityPath=1.000; Kuka.VelocityFieldEnabled=True; Kuka.ColDetectFieldEnabled=True; Kuka.CurrentCDSetIndex=0; Kuka.MovementParameterFieldEnabled=True; IlfCommand=SLIN
;ENDFOLD
SLIN XP629 WITH $VEL = SVEL_CP(2.0, , LCPDAT629),$TOOL = STOOL2(FP629),$BASE = SBASE(FP629.BASE_NO),$IPO_MODE = SIPO_MODE(FP629.IPO_FRAME),$LOAD = SLOAD(FP629.TOOL_NO),$ACC = SACC_CP(LCPDAT629),$ORI_TYPE = SORI_TYP(LCPDAT629),$APO = SAPO(LCPDAT629),$JERK = SJERK(LCPDAT629),$COLLMON_TOL_PRO[1] = USE_CM_PRO_VALUES(0)
;ENDFOLD

;FOLD SLIN P630 Vel=1 m/s CPDAT630 Tool[4]:Microflown3D Base[0];%{PE}
;FOLD Parameters ;%{h}
;Params IlfProvider=kukaroboter.basistech.inlineforms.movement.spline; Kuka.IsGlobalPoint=False; Kuka.PointName=P630; Kuka.BlendingEnabled=False; Kuka.MoveDataName=CPDAT630; Kuka.VelocityPath=1.000; Kuka.VelocityFieldEnabled=True; Kuka.ColDetectFieldEnabled=True; Kuka.CurrentCDSetIndex=0; Kuka.MovementParameterFieldEnabled=True; IlfCommand=SLIN
;ENDFOLD
SLIN XP630 WITH $VEL = SVEL_CP(2.0, , LCPDAT630),$TOOL = STOOL2(FP630),$BASE = SBASE(FP630.BASE_NO),$IPO_MODE = SIPO_MODE(FP630.IPO_FRAME),$LOAD = SLOAD(FP630.TOOL_NO),$ACC = SACC_CP(LCPDAT630),$ORI_TYPE = SORI_TYP(LCPDAT630),$APO = SAPO(LCPDAT630),$JERK = SJERK(LCPDAT630),$COLLMON_TOL_PRO[1] = USE_CM_PRO_VALUES(0)
;ENDFOLD

;FOLD SLIN P631 Vel=1 m/s CPDAT631 Tool[4]:Microflown3D Base[0];%{PE}
;FOLD Parameters ;%{h}
;Params IlfProvider=kukaroboter.basistech.inlineforms.movement.spline; Kuka.IsGlobalPoint=False; Kuka.PointName=P631; Kuka.BlendingEnabled=False; Kuka.MoveDataName=CPDAT631; Kuka.VelocityPath=1.000; Kuka.VelocityFieldEnabled=True; Kuka.ColDetectFieldEnabled=True; Kuka.CurrentCDSetIndex=0; Kuka.MovementParameterFieldEnabled=True; IlfCommand=SLIN
;ENDFOLD
SLIN XP631 WITH $VEL = SVEL_CP(2.0, , LCPDAT631),$TOOL = STOOL2(FP631),$BASE = SBASE(FP631.BASE_NO),$IPO_MODE = SIPO_MODE(FP631.IPO_FRAME),$LOAD = SLOAD(FP631.TOOL_NO),$ACC = SACC_CP(LCPDAT631),$ORI_TYPE = SORI_TYP(LCPDAT631),$APO = SAPO(LCPDAT631),$JERK = SJERK(LCPDAT631),$COLLMON_TOL_PRO[1] = USE_CM_PRO_VALUES(0)
;ENDFOLD

;FOLD SLIN P632 Vel=1 m/s CPDAT632 Tool[4]:Microflown3D Base[0];%{PE}
;FOLD Parameters ;%{h}
;Params IlfProvider=kukaroboter.basistech.inlineforms.movement.spline; Kuka.IsGlobalPoint=False; Kuka.PointName=P632; Kuka.BlendingEnabled=False; Kuka.MoveDataName=CPDAT632; Kuka.VelocityPath=1.000; Kuka.VelocityFieldEnabled=True; Kuka.ColDetectFieldEnabled=True; Kuka.CurrentCDSetIndex=0; Kuka.MovementParameterFieldEnabled=True; IlfCommand=SLIN
;ENDFOLD
SLIN XP632 WITH $VEL = SVEL_CP(2.0, , LCPDAT632),$TOOL = STOOL2(FP632),$BASE = SBASE(FP632.BASE_NO),$IPO_MODE = SIPO_MODE(FP632.IPO_FRAME),$LOAD = SLOAD(FP632.TOOL_NO),$ACC = SACC_CP(LCPDAT632),$ORI_TYPE = SORI_TYP(LCPDAT632),$APO = SAPO(LCPDAT632),$JERK = SJERK(LCPDAT632),$COLLMON_TOL_PRO[1] = USE_CM_PRO_VALUES(0)
;ENDFOLD

;FOLD SLIN P633 Vel=1 m/s CPDAT633 Tool[4]:Microflown3D Base[0];%{PE}
;FOLD Parameters ;%{h}
;Params IlfProvider=kukaroboter.basistech.inlineforms.movement.spline; Kuka.IsGlobalPoint=False; Kuka.PointName=P633; Kuka.BlendingEnabled=False; Kuka.MoveDataName=CPDAT633; Kuka.VelocityPath=1.000; Kuka.VelocityFieldEnabled=True; Kuka.ColDetectFieldEnabled=True; Kuka.CurrentCDSetIndex=0; Kuka.MovementParameterFieldEnabled=True; IlfCommand=SLIN
;ENDFOLD
SLIN XP633 WITH $VEL = SVEL_CP(2.0, , LCPDAT633),$TOOL = STOOL2(FP633),$BASE = SBASE(FP633.BASE_NO),$IPO_MODE = SIPO_MODE(FP633.IPO_FRAME),$LOAD = SLOAD(FP633.TOOL_NO),$ACC = SACC_CP(LCPDAT633),$ORI_TYPE = SORI_TYP(LCPDAT633),$APO = SAPO(LCPDAT633),$JERK = SJERK(LCPDAT633),$COLLMON_TOL_PRO[1] = USE_CM_PRO_VALUES(0)
;ENDFOLD

;FOLD SLIN P634 Vel=1 m/s CPDAT634 Tool[4]:Microflown3D Base[0];%{PE}
;FOLD Parameters ;%{h}
;Params IlfProvider=kukaroboter.basistech.inlineforms.movement.spline; Kuka.IsGlobalPoint=False; Kuka.PointName=P634; Kuka.BlendingEnabled=False; Kuka.MoveDataName=CPDAT634; Kuka.VelocityPath=1.000; Kuka.VelocityFieldEnabled=True; Kuka.ColDetectFieldEnabled=True; Kuka.CurrentCDSetIndex=0; Kuka.MovementParameterFieldEnabled=True; IlfCommand=SLIN
;ENDFOLD
SLIN XP634 WITH $VEL = SVEL_CP(2.0, , LCPDAT634),$TOOL = STOOL2(FP634),$BASE = SBASE(FP634.BASE_NO),$IPO_MODE = SIPO_MODE(FP634.IPO_FRAME),$LOAD = SLOAD(FP634.TOOL_NO),$ACC = SACC_CP(LCPDAT634),$ORI_TYPE = SORI_TYP(LCPDAT634),$APO = SAPO(LCPDAT634),$JERK = SJERK(LCPDAT634),$COLLMON_TOL_PRO[1] = USE_CM_PRO_VALUES(0)
;ENDFOLD

;FOLD SLIN P635 Vel=1 m/s CPDAT635 Tool[4]:Microflown3D Base[0];%{PE}
;FOLD Parameters ;%{h}
;Params IlfProvider=kukaroboter.basistech.inlineforms.movement.spline; Kuka.IsGlobalPoint=False; Kuka.PointName=P635; Kuka.BlendingEnabled=False; Kuka.MoveDataName=CPDAT635; Kuka.VelocityPath=1.000; Kuka.VelocityFieldEnabled=True; Kuka.ColDetectFieldEnabled=True; Kuka.CurrentCDSetIndex=0; Kuka.MovementParameterFieldEnabled=True; IlfCommand=SLIN
;ENDFOLD
SLIN XP635 WITH $VEL = SVEL_CP(2.0, , LCPDAT635),$TOOL = STOOL2(FP635),$BASE = SBASE(FP635.BASE_NO),$IPO_MODE = SIPO_MODE(FP635.IPO_FRAME),$LOAD = SLOAD(FP635.TOOL_NO),$ACC = SACC_CP(LCPDAT635),$ORI_TYPE = SORI_TYP(LCPDAT635),$APO = SAPO(LCPDAT635),$JERK = SJERK(LCPDAT635),$COLLMON_TOL_PRO[1] = USE_CM_PRO_VALUES(0)
;ENDFOLD

;FOLD SLIN P636 Vel=1 m/s CPDAT636 Tool[4]:Microflown3D Base[0];%{PE}
;FOLD Parameters ;%{h}
;Params IlfProvider=kukaroboter.basistech.inlineforms.movement.spline; Kuka.IsGlobalPoint=False; Kuka.PointName=P636; Kuka.BlendingEnabled=False; Kuka.MoveDataName=CPDAT636; Kuka.VelocityPath=1.000; Kuka.VelocityFieldEnabled=True; Kuka.ColDetectFieldEnabled=True; Kuka.CurrentCDSetIndex=0; Kuka.MovementParameterFieldEnabled=True; IlfCommand=SLIN
;ENDFOLD
SLIN XP636 WITH $VEL = SVEL_CP(2.0, , LCPDAT636),$TOOL = STOOL2(FP636),$BASE = SBASE(FP636.BASE_NO),$IPO_MODE = SIPO_MODE(FP636.IPO_FRAME),$LOAD = SLOAD(FP636.TOOL_NO),$ACC = SACC_CP(LCPDAT636),$ORI_TYPE = SORI_TYP(LCPDAT636),$APO = SAPO(LCPDAT636),$JERK = SJERK(LCPDAT636),$COLLMON_TOL_PRO[1] = USE_CM_PRO_VALUES(0)
;ENDFOLD

;FOLD SLIN P637 Vel=1 m/s CPDAT637 Tool[4]:Microflown3D Base[0];%{PE}
;FOLD Parameters ;%{h}
;Params IlfProvider=kukaroboter.basistech.inlineforms.movement.spline; Kuka.IsGlobalPoint=False; Kuka.PointName=P637; Kuka.BlendingEnabled=False; Kuka.MoveDataName=CPDAT637; Kuka.VelocityPath=1.000; Kuka.VelocityFieldEnabled=True; Kuka.ColDetectFieldEnabled=True; Kuka.CurrentCDSetIndex=0; Kuka.MovementParameterFieldEnabled=True; IlfCommand=SLIN
;ENDFOLD
SLIN XP637 WITH $VEL = SVEL_CP(2.0, , LCPDAT637),$TOOL = STOOL2(FP637),$BASE = SBASE(FP637.BASE_NO),$IPO_MODE = SIPO_MODE(FP637.IPO_FRAME),$LOAD = SLOAD(FP637.TOOL_NO),$ACC = SACC_CP(LCPDAT637),$ORI_TYPE = SORI_TYP(LCPDAT637),$APO = SAPO(LCPDAT637),$JERK = SJERK(LCPDAT637),$COLLMON_TOL_PRO[1] = USE_CM_PRO_VALUES(0)
;ENDFOLD

;FOLD SLIN P638 Vel=1 m/s CPDAT638 Tool[4]:Microflown3D Base[0];%{PE}
;FOLD Parameters ;%{h}
;Params IlfProvider=kukaroboter.basistech.inlineforms.movement.spline; Kuka.IsGlobalPoint=False; Kuka.PointName=P638; Kuka.BlendingEnabled=False; Kuka.MoveDataName=CPDAT638; Kuka.VelocityPath=1.000; Kuka.VelocityFieldEnabled=True; Kuka.ColDetectFieldEnabled=True; Kuka.CurrentCDSetIndex=0; Kuka.MovementParameterFieldEnabled=True; IlfCommand=SLIN
;ENDFOLD
SLIN XP638 WITH $VEL = SVEL_CP(2.0, , LCPDAT638),$TOOL = STOOL2(FP638),$BASE = SBASE(FP638.BASE_NO),$IPO_MODE = SIPO_MODE(FP638.IPO_FRAME),$LOAD = SLOAD(FP638.TOOL_NO),$ACC = SACC_CP(LCPDAT638),$ORI_TYPE = SORI_TYP(LCPDAT638),$APO = SAPO(LCPDAT638),$JERK = SJERK(LCPDAT638),$COLLMON_TOL_PRO[1] = USE_CM_PRO_VALUES(0)
;ENDFOLD

;FOLD SLIN P639 Vel=1 m/s CPDAT639 Tool[4]:Microflown3D Base[0];%{PE}
;FOLD Parameters ;%{h}
;Params IlfProvider=kukaroboter.basistech.inlineforms.movement.spline; Kuka.IsGlobalPoint=False; Kuka.PointName=P639; Kuka.BlendingEnabled=False; Kuka.MoveDataName=CPDAT639; Kuka.VelocityPath=1.000; Kuka.VelocityFieldEnabled=True; Kuka.ColDetectFieldEnabled=True; Kuka.CurrentCDSetIndex=0; Kuka.MovementParameterFieldEnabled=True; IlfCommand=SLIN
;ENDFOLD
SLIN XP639 WITH $VEL = SVEL_CP(2.0, , LCPDAT639),$TOOL = STOOL2(FP639),$BASE = SBASE(FP639.BASE_NO),$IPO_MODE = SIPO_MODE(FP639.IPO_FRAME),$LOAD = SLOAD(FP639.TOOL_NO),$ACC = SACC_CP(LCPDAT639),$ORI_TYPE = SORI_TYP(LCPDAT639),$APO = SAPO(LCPDAT639),$JERK = SJERK(LCPDAT639),$COLLMON_TOL_PRO[1] = USE_CM_PRO_VALUES(0)
;ENDFOLD

;FOLD SLIN P640 Vel=1 m/s CPDAT640 Tool[4]:Microflown3D Base[0];%{PE}
;FOLD Parameters ;%{h}
;Params IlfProvider=kukaroboter.basistech.inlineforms.movement.spline; Kuka.IsGlobalPoint=False; Kuka.PointName=P640; Kuka.BlendingEnabled=False; Kuka.MoveDataName=CPDAT640; Kuka.VelocityPath=1.000; Kuka.VelocityFieldEnabled=True; Kuka.ColDetectFieldEnabled=True; Kuka.CurrentCDSetIndex=0; Kuka.MovementParameterFieldEnabled=True; IlfCommand=SLIN
;ENDFOLD
SLIN XP640 WITH $VEL = SVEL_CP(2.0, , LCPDAT640),$TOOL = STOOL2(FP640),$BASE = SBASE(FP640.BASE_NO),$IPO_MODE = SIPO_MODE(FP640.IPO_FRAME),$LOAD = SLOAD(FP640.TOOL_NO),$ACC = SACC_CP(LCPDAT640),$ORI_TYPE = SORI_TYP(LCPDAT640),$APO = SAPO(LCPDAT640),$JERK = SJERK(LCPDAT640),$COLLMON_TOL_PRO[1] = USE_CM_PRO_VALUES(0)
;ENDFOLD

